# B&R Automation Studio project NAEUL004C00R13L518F00 (part 33)

#### Act_Main.st - Do Not Change!!!
```iecst
(** 2020-10-05 **)
ACTION Act_Main:
	//Reset Done
	IF tylocalHWInfo.Out.eStatus = Done AND tylocalHWInfo.In.eAct = HWInfoActIdle THEN
		tylocalHWInfo.Out.eStat	:= HWInfoActIdle;
	END_IF

	//Set tylocalHWInfo.In.eAct
	IF tylocalHWInfo.Out.eStatus = Idle THEN
		tylocalHWInfo.Out.eStat	:= tylocalHWInfo.In.eAct;
	END_IF

	//Main
	CASE tylocalHWInfo.Out.eStat OF

		HWInfoActIdle:
			IF tylocalHWInfo.Out.eStatus <> Idle THEN	//Reset Data
				//Private
				fbGetIPAddr(enable := FALSE);
				fbGetMacAddr(enable := FALSE);
				fbSetIPAddr(enable := FALSE);
				fbSetSubnetMask(enable := FALSE);
				fbGetETHConfigMode(enable := FALSE);
				fbSetETHConfigMode(enable := FALSE);

				tylocalHWInfo.Out.sStatTxt	:= a_sStatText[tylocalHWInfo.Out.eStat];

			END_IF

			tylocalHWInfo.Out.eStatus	:= Idle;

		HWInfoActGetIPAddr:
			IF tylocalHWInfo.Out.eStatus = Idle OR tylocalHWInfo.Out.eStatus = Busy THEN

				tylocalHWInfo.Out.eStatus	:= Busy;

				tylocalHWInfo.Out.sStatTxt	:= a_sStatText[tylocalHWInfo.Out.eStat];

				IF DiagCpuIsSimulated() = FALSE THEN
					fbGetIPAddr(enable := TRUE);
					IF fbGetIPAddr.status = 0 THEN
						tylocalHWInfo.Out.eStatus	:= Done;
					ELSIF fbGetIPAddr.status < 65534 THEN
						udiStatus	:= 10000;	//Get IP Address Error
						tylocalHWInfo.Out.eStatus		:= Error;
					END_IF

				ELSE
					tylocalHWInfo.Out.eStatus	:= Done;
					tylocalHWInfo.Out.sIPAddr	:= '127.0.0.1';

				END_IF

			END_IF

		HWInfoActGetSubnetMask:
			IF tylocalHWInfo.Out.eStatus = Idle OR tylocalHWInfo.Out.eStatus = Busy THEN

				tylocalHWInfo.Out.eStatus	:= Busy;

				tylocalHWInfo.Out.sStatTxt	:= a_sStatText[tylocalHWInfo.Out.eStat];

				IF DiagCpuIsSimulated() = FALSE THEN
					fbGetSubnetMask(enable := TRUE);
					IF fbGetSubnetMask.status = 0 THEN
						tylocalHWInfo.Out.eStatus	:= Done;
					ELSIF fbGetSubnetMask.status < 65534 THEN
						udiStatus	:= 10001;	//Get Subnet Mask Error
						tylocalHWInfo.Out.eStatus		:= Error;
					END_IF

				ELSE
					tylocalHWInfo.Out.eStatus		:= Done;
					tylocalHWInfo.Out.sSubnetMask	:= '255.255.0.0';

				END_IF

			END_IF

		HWInfoActGetMacAddr:
			IF tylocalHWInfo.Out.eStatus = Idle OR tylocalHWInfo.Out.eStatus = Busy THEN

				tylocalHWInfo.Out.eStatus	:= Busy;

				tylocalHWInfo.Out.sStatTxt	:= a_sStatText[tylocalHWInfo.Out.eStat];

				IF DiagCpuIsSimulated() = FALSE THEN
					fbGetMacAddr(enable := TRUE);
					IF fbGetMacAddr.status = 0 THEN
						tylocalHWInfo.Out.eStatus	:= Done;
					ELSIF fbGetMacAddr.status < 65534 THEN
						udiStatus	:= 10002;	//Get Mac Address Error
						tylocalHWInfo.Out.eStatus		:= Error;
					END_IF

				ELSE
					tylocalHWInfo.Out.eStatus	:= Done;

				END_IF

			END_IF

		HWInfoActSetIPAddr:
			IF tylocalHWInfo.Out.eStatus = Idle OR tylocalHWInfo.Out.eStatus = Busy THEN

				tylocalHWInfo.Out.eStatus	:= Busy;

				tylocalHWInfo.Out.sStatTxt	:= a_sStatText[tylocalHWInfo.Out.eStat];

				IF DiagCpuIsSimulated() = FALSE THEN
					fbSetIPAddr(enable := TRUE);
					IF fbSetIPAddr.status = 0 THEN
						tylocalHWInfo.Out.sIPAddr	:= p_sSetIPAddr;
						tylocalHWInfo.Out.eStatus	:= Done;
					ELSIF fbSetIPAddr.status < 65534 THEN
						udiStatus	:= 10003;	//Set IP Address Error
						tylocalHWInfo.Out.eStatus		:= Error;
					END_IF

				ELSE
					tylocalHWInfo.Out.eStatus	:= Done;

				END_IF

			END_IF

		HWInfoActSetSubnetMask:
			IF tylocalHWInfo.Out.eStatus = Idle OR tylocalHWInfo.Out.eStatus = Busy THEN

				tylocalHWInfo.Out.eStatus	:= Busy;

				tylocalHWInfo.Out.sStatTxt	:= a_sStatText[tylocalHWInfo.Out.eStat];

				IF DiagCpuIsSimulated() = FALSE THEN
					fbSetSubnetMask(enable := TRUE);
					IF fbSetSubnetMask.status = 0 THEN
						tylocalHWInfo.Out.sSubnetMask	:= p_sSetSubnetMask;
						tylocalHWInfo.Out.eStatus		:= Done;
					ELSIF fbSetSubnetMask.status < 65534 THEN
						udiStatus	:= 10004;	//Set Subnet Mask Error
						tylocalHWInfo.Out.eStatus		:= Error;
					END_IF

				ELSE
					tylocalHWInfo.Out.eStatus	:= Done;

				END_IF

			END_IF

		HWInfoActGetEthConfigMode:
			IF tylocalHWInfo.Out.eStatus = Idle OR tylocalHWInfo.Out.eStatus = Busy THEN

				tylocalHWInfo.Out.eStatus	:= Busy;

				tylocalHWInfo.Out.sStatTxt	:= a_sStatText[tylocalHWInfo.Out.eStat];
				IF DiagCpuIsSimulated() = FALSE THEN
					fbGetETHConfigMode(enable := TRUE);
					IF fbGetETHConfigMode.status = 0 THEN
						tylocalHWInfo.Out.udiConfigMode := fbGetETHConfigMode.ConfigMode;
						tylocalHWInfo.Out.eStatus	:= Done;
					ELSIF fbGetETHConfigMode.status < 65534 THEN
						udiStatus	:= 10005;	//Get Network Configuration  Error
						tylocalHWInfo.Out.eStatus		:= Error;
					END_IF

				ELSE
					tylocalHWInfo.Out.eStatus	:= Done;

				END_IF

			END_IF

		HWInfoActSetEthConfigMode:
			IF tylocalHWInfo.Out.eStatus = Idle OR tylocalHWInfo.Out.eStatus = Busy THEN

				tylocalHWInfo.Out.eStatus	:= Busy;

				tylocalHWInfo.Out.sStatTxt	:= a_sStatText[tylocalHWInfo.Out.eStat];

				IF DiagCpuIsSimulated() = FALSE THEN
					fbSetETHConfigMode.ConfigMode := USINT_TO_UDINT(p_usiNetworkMod);
					fbSetETHConfigMode(enable := TRUE);

					IF fbSetETHConfigMode.status = 0 THEN
						tylocalHWInfo.Out.eStatus	:= Done;
					ELSIF fbSetETHConfigMode.status < 65534 THEN
						udiStatus	:= 10006;	//Set Network Configuration  Error
						tylocalHWInfo.Out.eStatus		:= Error;
					END_IF

				ELSE
					tylocalHWInfo.Out.eStatus	:= Done;

				END_IF

			END_IF

		HWInfoActSetDefaultGateway:
			IF tylocalHWInfo.Out.eStatus = Idle OR tylocalHWInfo.Out.eStatus = Busy THEN

				tylocalHWInfo.Out.eStatus	:= Busy;

				tylocalHWInfo.Out.sStatTxt	:= a_sStatText[tylocalHWInfo.Out.eStat];

				IF DiagCpuIsSimulated() = FALSE THEN
					fbSetDefaultGateway.pGateway := ADR(p_sSetDefaultGW);
					fbSetDefaultGateway(enable := TRUE);

					IF fbSetDefaultGateway.status = 0 THEN
						tylocalHWInfo.Out.eStatus	:= Done;
					ELSIF fbSetDefaultGateway.status < 65534 THEN
						udiStatus	:= 10007;	//'Set Default Gateway IP Error'
						tylocalHWInfo.Out.eStatus		:= Error;
					END_IF

				ELSE
					tylocalHWInfo.Out.eStatus	:= Done;
				END_IF

			END_IF

	END_CASE

	//Generate file
//	IF tylocalHWInfo.Out.a_usiMacAddr[3] <> 0 AND usiInitialFile <2 THEN
//		CASE usi OF
//			0:
//				FOR usi:= 0 TO 5 DO
//					//a_sMacAddr[usi] := USINT_TO_STRING(tylocalHWInfo.Out.a_usiMacAddr[usi]);
//					sprintf1(ADR(a_sMacAddr[usi]), ADR('%+02x'), tylocalHWInfo.Out.a_usiMacAddr[usi]);
//				END_FOR
//				sMacAddr := CONCAT('PLC= ',CONCAT(a_sMacAddr[0],'-'));
//				FOR usi := 1 TO 5 DO
//					sMacAddr := CONCAT(CONCAT(sMacAddr,a_sMacAddr[usi]),'-');
//				END_FOR
//				sMacAddr := DELETE(sMacAddr,1,LEN(sMacAddr));
//				usi := 1;
//			1:
//				fbFileFullWrite_0(bEn := TRUE, sDevice := 'Log', sFile := 'PLC_MacAddress.txt', udiOffset := 0, p_Src := ADR(sMacAddr), udiLen := SIZEOF(sMacAddr), udiOption := 0);
//				IF fbFileFullWrite_0.udiStatus = 0 THEN
//					fbFileFullWrite_0(bEn := FALSE);
//					IF usiInitialFile = 1 THEN
//						usi := 0;
//					END_IF
//					usiInitialFile := usiInitialFile +1;
//				END_IF
//
//		END_CASE
//	END_IF
END_ACTION
```

#### Act_Alarm.st - Do Not Change!!!
```iecst
(** 2019-03-25 **)
ACTION Act_Alarm:
	IF tylocalHWInfo.In.udiRstErr <> udiRstErrOld THEN
		bRstErr			:= TRUE;
		udiRstErrOld	:= tylocalHWInfo.In.udiRstErr;
	ELSE
		bRstErr			:= FALSE;
	END_IF

	//Reset Error
	IF (tylocalHWInfo.Out.eStatus = Error) AND bRstErr THEN
		tylocalHWInfo.In.eAct	:= HWInfoActIdle;
		tylocalHWInfo.Out.eStat	:= HWInfoActIdle;
	END_IF

	//Error
	IF EDGEPOS(tylocalHWInfo.Out.eStatus = Error) THEN

		tylocalHWInfo.Out.tyAlmData.udiCode			:= udiStatus;
		tylocalHWInfo.Out.tyAlmData.eSeverity		:= AlmSeverityError;
		tylocalHWInfo.Out.tyAlmData.udiRunTime		:= tylocalHWInfo.Out.tyAlmData.udiRunTime + 1;
		tylocalHWInfo.Out.tyAlmData.bAlm			:= TRUE;
		tylocalHWInfo.Out.tyAlmData.udiModuleNum	:= udiModuleNum;
		g_tyAlmProgNm.sHWinfoProgNm					:= tylocalHWInfo.In.sProgNm;

	ELSIF bRstErr AND (tylocalHWInfo.Out.tyAlmData.udiCode <> 0) THEN

		tylocalHWInfo.Out.tyAlmData.udiCode		:= 0;
		tylocalHWInfo.Out.tyAlmData.eSeverity	:= AlmSeverityNA;
		tylocalHWInfo.Out.tyAlmData.bAlm		:= FALSE;

		tylocalHWInfo.Out.sStatTxt	:= a_sStatText[tylocalHWInfo.Out.eStat];

	END_IF

END_ACTION
```

#### Local.var - Do Not Change!!!
```iecst
(*2020-09-22*)
VAR
	tylocalHWInfo : tyHWInfo;
END_VAR
(**)
(*Local Action, State & Status*)
VAR
	eStatus : eFBStatus := Idle;
	udiStatus : UDINT := 0;
	sStatTxt : STRING[200] := '';
	a_sStatText : ARRAY[0..50] OF STRING[200] := ['Idling','Get IP Address','Get IP Subnet Mask','Get Mac Address','Setting IP Address','Setting IP Subnet Mask',45('')];
END_VAR
(**)
(*Local Alarm*)
VAR
	tyAlmData : tyAlmDat;
	a_tyAlmText : ARRAY[10000..10099] OF tyAlmTxt := [(sAlmText:='Get IP Address Error',sRcyText:='Failed To Obtain The IP Address. Please Contact Nutek For A Possible Solution.'),(sAlmText:='Get Subnet Mask Error',sRcyText:='Failed To Obtain The Subnet Mask. Please Contact Nutek For A Possible Solution.'),(sAlmText:='Get Mac Address Error',sRcyText:='Failed To Obtain The Mac Address. Please Contact Nutek For A Possible Solution.'),(sAlmText:='Set IP Address Error',sRcyText:='Invalid IP Address Configuration. Please Contact Nutek For A Possible Solution.'),(sAlmText:='Set Subnet Mask Error',sRcyText:='Invalid Subnet Mask Configuration. Please Contact Nutek For A Possible Solution.'),(sAlmText:='Get Network Configuration Mode Error',sRcyText:='Failed To Obtain The Network Configuration. Please Contact Nutek For A Possible Solution.'),(sAlmText:='Set Network Configuration Mode Error',sRcyText:='Invalid Network Configuration . Please Contact Nutek For A Possible Solution.'),(sAlmText:='Set Default Gateway IP Error',sRcyText:='Invalid IP Address Configuration. Please Contact Nutek For A Possible Solution.'),92((0))];
END_VAR
(**)
(*Local Output*)
VAR
	sIPAddr : STRING[15];
	sSubnetMask : STRING[15];
	a_usiMacAddr : ARRAY[0..5] OF USINT;
	udiConfigMode : UDINT;
END_VAR
(**)
(*Local Input*)
VAR
	udiRstErr : UDINT := 0;
	sSetIPAddr : STRING[15];
	sSetSubnetMask : STRING[15];
	sDevice : STRING[3] := 'IF2';
	sProgNm : STRING[15] := 'HWInfo';
	bNtSettingsLoadDone : BOOL := TRUE;
	usiNetworkMode : USINT;
	sSetDefaultGW : STRING[15];
END_VAR
(**)
(*Local*)
VAR
	bRstErr : BOOL;
	udiRstErrOld : UDINT;
	bInitDone : BOOL;
	bInitialDone : BOOL;
	fbGetIPAddr : CfgGetIPAddr;
	fbGetSubnetMask : CfgGetSubnetMask;
	fbGetMacAddr : CfgGetMacAddr;
	fbSetIPAddr : CfgSetIPAddr;
	fbSetSubnetMask : CfgSetSubnetMask;
	fbSetETHConfigMode : CfgSetEthConfigMode;
	fbGetETHConfigMode : CfgGetEthConfigMode;
	fbSetDefaultGateway : CfgSetDefaultGateway;
	udiModuleNum : UDINT := 5651;
END_VAR
(**)
(*MAC Address*)
VAR
	sMacAddress : tysMacAddress;
END_VAR
(**)
VAR
	sPLCMacAddress : STRING[27];
	sHMIMacAddress : STRING[27];
END_VAR
```

#### InputRef.var - not listed in the package file held
```iecst
(*2020-09-22*)
(**)
(*General*)
VAR
	p_eAct : REFERENCE TO eHWInfoAction;
	p_udiRstErr : REFERENCE TO UDINT;
END_VAR
(**)
(*Configuration*)
VAR
	p_sSetIPAddr : REFERENCE TO STRING[15];
	p_sSetSubnetMask : REFERENCE TO STRING[15];
	p_sDevice : REFERENCE TO STRING[3];
	p_sProgNm : REFERENCE TO STRING[15];
	p_bNtSettingsLoadDone : REFERENCE TO BOOL;
	p_usiNetworkMod : REFERENCE TO USINT;
	p_sSetDefaultGW : REFERENCE TO STRING[15];
END_VAR
```

#### InputRef_Link.var - not listed in the package file held
```iecst
(*2019-03-25*)
(**)
VAR
	p_bLinkStartupRun : REFERENCE TO BOOL;
	p_sHMIMacAdd : REFERENCE TO STRING[27];
END_VAR
```

#### Act_InitGlobal.st - not listed in the package file held
```iecst
(** 2020-09-22 **)
ACTION Act_InitGlobal:

	(* Always Change If Project Change *)

	//Pass Data To Link
	p_bLinkStartupRun ACCESS p_StartupRun;

	//Pass Data To Internal Use
	p_udiRstErr ACCESS p_RstErrReset;
	p_sSetIPAddr ACCESS p_UISetIPAddr;
	p_sSetSubnetMask ACCESS p_UISetSubnetMask;
	p_sDevice ACCESS p_NtParamHWInfoDevice;
	p_sProgNm ACCESS p_NtParamHWInfoProgNm;
	p_bNtSettingsLoadDone ACCESS p_StartupNtSettingsLoadDone;
	p_usiNetworkMod ACCESS p_UINetworkMode;

	//HMI MAC Address
	p_sHMIMacAdd ACCESS p_NtParamHWInfoHMIMacAddress;
	p_sSetDefaultGW ACCESS p_McParamDefaultGateway;

	(* Always Change If Project Change *)

END_ACTION
```

#### Act_InitLocal.st - not listed in the package file held
```iecst
(** 2020-09-22 **)
ACTION Act_InitLocal:

	//Input Reference Link To Local Variable
	p_eAct ACCESS ADR(eAct);
	p_udiRstErr ACCESS ADR(udiRstErr);
	p_sSetIPAddr ACCESS ADR(sSetIPAddr);
	p_sSetSubnetMask ACCESS ADR(sSetSubnetMask);
	p_sDevice ACCESS ADR(sDevice);
	p_sProgNm ACCESS ADR(sProgNm);
	p_bNtSettingsLoadDone ACCESS ADR(bNtSettingsLoadDone);
	p_usiNetworkMod ACCESS ADR(usiNetworkMode);
	p_sSetDefaultGW ACCESS ADR(sSetDefaultGW);
END_ACTION
```

### TLBuz.typ - Do Not Change!!!
```iecst
(*2020-02-19*)
(**)
(*Action*)

TYPE
	eTLBuzAction :
		(
		TLBuzActIdle,
		TLBuzActSetGreen,
		TLBuzActSetWhite,
		TLBuzActSetRed,
		TLBuzActSetAmber,
		TLBuzActSetBlue,
		TLBuzActSetBuz,
		TLBuzActRstGreen,
		TLBuzActRstWhite,
		TLBuzActRstRed,
		TLBuzActRstAmber,
		TLBuzActRstBlue,
		TLBuzActRstBuz,
		TLBuzActSetAll,
		TLBuzActRstAll
		);
	eTLBuzMod :
		(
		TLBuzModNutek,
		TLBuzModAptiv,
		TLBuzModMEK,
		TLBuzModBHTC,
		TLBuzModSiemens_2Colour
		);
	tyTLBuz : 	STRUCT
		In : tyTLBuzIn1;
		Out : tyTLBuzOut1;
	END_STRUCT;
	tyTLBuzIn1 : 	STRUCT
		eAct : eTLBuzAction; (*Tower Light Buzzer's Action*)
		bCoverSwitchSig : BOOL := FALSE; (*Cover Switch Signal*)
		bAOIErrSig : BOOL := FALSE; (*AOI Err Signal*)
		bAOIOriginSig : BOOL := FALSE; (*AOI Origin Signal*)
		bBuzAlertEn : BOOL := FALSE; (*Buzzer Alert Enable*)
		bTLBlueFlashEn : BOOL := FALSE; (*Tower Light Blue Flash Enable*)
		bTLAmberFlashEn : BOOL := FALSE; (*Tower Light Amber Flash Enable*)
		bTLWhiteFlashEn : BOOL := FALSE; (*Tower Light White Flash Enable*)
		bTLRedFlashEn : BOOL := FALSE; (*Tower Light Red Flash Enable*)
		bTLGreenFlashEn : BOOL := FALSE; (*Tower Light Green Flash Enable*)
		bUIManualMod : BOOL := FALSE; (*Manual Mode*)
		bStartup : BOOL := FALSE; (*Startup Mode*)
		bErr : BOOL := FALSE; (*Error Exist*)
		bErrNoBuz : BOOL := FALSE; (*Error Exist With No Buzzer*)
		bWarning : ARRAY[0..5]OF BOOL := [6(FALSE)]; (*Warning*)
		bWarningNoBuz : ARRAY[0..5]OF BOOL := [6(FALSE)]; (*Warning With No Buzzer*)
		bChgRcp : BOOL := FALSE; (*Change Recipe*)
		bSeqStop : BOOL := FALSE; (*Sequence Stop*)
		bStep : BOOL := FALSE; (*Step*)
		bOps : BOOL := FALSE; (*Operation Mode*)
		bStandby : BOOL := FALSE; (*Standby Mode*)
		bSimulation : BOOL := FALSE; (*Simulation Mode*)
		bMuteBuz : BOOL := FALSE; (*Mute Buzzer*)
		tTLChgRcpBlinkTm : TIME := T#200ms; (*Tower Light Change Recipe Blink Timer*)
		tTLErrBlinkTm : TIME := T#500ms; (*Tower Light Error Blink Timer*)
		tBuzErrOnTm : TIME := T#500ms; (*Buzzer Error On Timer*)
		tBuzErrRestTm : TIME := T#500ms; (*Buzzer Error Reset Timer*)
		usiBuzErrOnCntr : USINT := 3; (*Buzzer Error On Counter*)
		bBuzErrStopSeqEn : BOOL := FALSE; (*Buzzer Error Stop Sequence Timer Counter*)
		usiBuzErrStopSeqCntr : USINT := 3; (*Buzzer Error Stop Sequence Counter*)
		tTLWarnBlinkTm : ARRAY[0..5]OF TIME := [6(T#500ms)]; (*Tower Light Warning Blink Timer*)
		tBuzWarnOnTm : ARRAY[0..5]OF TIME := [6(T#500ms)]; (*Buzzer Warning On Timer*)
		tBuzWarnRestTm : ARRAY[0..5]OF TIME := [6(T#5s)]; (*Buzzer Warning Reset Timer*)
		usiBuzWarnOnCntr : ARRAY[0..5]OF USINT := [6(3)]; (*Buzzer Warning On Counter*)
		bBuzWarnStopSeqEn : ARRAY[0..5]OF BOOL := [6(FALSE)]; (*Buzzer Warning Stop Sequence Enable*)
		usiBuzWarnStopSeqCntr : ARRAY[0..5]OF USINT := [6(3)]; (*Buzzer Warning Stop Sequence Counter*)
		tTLWarn1BlinkTm : TIME := T#500ms;
		tBuzWarn1OnTm : TIME := T#500ms;
		tBuzWarn1RestTm : TIME := T#5s;
		usiBuzWarn1OnCntr : USINT := 3;
		bBuzWarn1StopSeqEn : BOOL := FALSE;
		usiBuzWarn1StopSeqCntr : USINT := 3;
		tTLWarn2BlinkTm : TIME := T#500ms;
		tBuzWarn2OnTm : TIME := T#500ms;
		tBuzWarn2RestTm : TIME := T#5s;
		usiBuzWarn2OnCntr : USINT := 3;
		bBuzWarn2StopSeqEn : BOOL := FALSE;
		usiBuzWarn2StopSeqCntr : USINT := 3;
		tTLWarn3BlinkTm : TIME := T#500ms;
		tBuzWarn3OnTm : TIME := T#500ms;
		tBuzWarn3RestTm : TIME := T#5s;
		usiBuzWarn3OnCntr : USINT := 3;
		bBuzWarn3StopSeqEn : BOOL := FALSE;
		usiBuzWarn3StopSeqCntr : USINT := 3;
		tTLWarn4BlinkTm : TIME := T#500ms;
		tBuzWarn4OnTm : TIME := T#500ms;
		tBuzWarn4RestTm : TIME := T#5s;
		usiBuzWarn4OnCntr : USINT := 3;
		bBuzWarn4StopSeqEn : BOOL := FALSE;
		usiBuzWarn4StopSeqCntr : USINT := 3;
		tTLWarn5BlinkTm : TIME := T#500ms;
		tBuzWarn5OnTm : TIME := T#500ms;
		tBuzWarn5RestTm : TIME := T#5s;
		usiBuzWarn5OnCntr : USINT := 3;
		bBuzWarn5StopSeqEn : BOOL := FALSE;
		usiBuzWarn5StopSeqCntr : USINT := 3;
		tBuzAlertOnTm : TIME := T#500ms; (*Buzzer Alert On Timer*)
		tBuzAlertRestTm : TIME := T#5s; (*Buzzer Alert Reset Timer*)
		usiBuzAlertOnCntr : USINT := 3; (*Buzzer Alert On Counter*)
		bBuzAlertStopSeqEn : BOOL := FALSE; (*Buzzer Alert Stop Sequence Enable*)
		usiBuzAlertStopSeqCntr : USINT := 3; (*Buzzer Alert Stop Sequence Counter*)
		tTLBlueBlinkTm : TIME := T#500ms; (*Tower Light Blue Blink Timer*)
		tTLAmberBlinkTm : TIME := T#500ms; (*Tower Light Amber Blink Timer*)
		tTLWhiteBlinkTm : TIME := T#500ms; (*Tower Light White Blink Timer*)
		tTLRedBlinkTm : TIME := T#500ms; (*Tower Light Red Blink Timer*)
		tTLGreenBlinkTm : TIME := T#500ms; (*Tower Light Green Blink Timer*)
		eTLBuzMode : eTLBuzMod := TLBuzModNutek; (*Tower Light Buzzer Mode*)
		bMcParamAGVComEn : BOOL;
		eMcParamMagExMode : eMcMagExchangeMode;
	END_STRUCT;
	tyTLBuzOut1 : 	STRUCT
		eStat : eTLBuzAction := TLBuzActIdle; (*Tower Light Buzzer's State*)
		eStatus : eFBStatus := Idle; (*Tower Light Buzzer's Status*)
		sStatTxt : STRING[200] := ''; (*Tower Light Buzzer's State in Text*)
		bTLBlue : BOOL; (*Tower Light Blue*)
		bTLRed : BOOL; (*Tower Light Red*)
		bTLAmber : BOOL; (*Tower Light Amber*)
		bTLWhite : BOOL; (*Tower Light White*)
		bTLGreen : BOOL; (*Tower Light Green*)
		bBuzBeep : BOOL; (*Buzzer Beeping*)
	END_STRUCT;
END_TYPE
```

### TLBuz.var - Change By Project
```iecst
(*2019-03-25*)
VAR
	g_tyTLBuz : tyTLBuzOut1;
END_VAR
(**)
```

### Program Logical/TLBuz/TLBuz (IEC, version 1.00.0) - 1.00.0 - NtTLBuz v5.00.0

#### Act_InputConfig.st - Change By Project
```iecst
ACTION Act_InputConfig:

	tylocalTLBuz.In.bStartup 					:= g_tyStartUp.bRun;
	tylocalTLBuz.In.bErr	 					:= g_tyAlm.bErr;
	tylocalTLBuz.In.bSeqStop    				:= g_tyOps.bStatusCycleStop;
	tylocalTLBuz.In.bStep						:= g_tyOps.bStatusStep;
	tylocalTLBuz.In.bOps						:= g_tyOps.bStatusRun;
	tylocalTLBuz.In.bStandby					:= g_tyOps.bStatusStop;
	tylocalTLBuz.In.bMuteBuz					:= g_tyUIOut.bUIMuteBuz;
	tylocalTLBuz.In.bUIManualMod				:= g_tyUIOut.bUIManualMod;

	//  -----------------------------------------  TLBuz 5.00.2  -----------------------------------------	//

	tylocalTLBuz.In.tTLChgRcpBlinkTm 			:= g_tyNtParamCurr.tyTLBuz.tTLChgRcpBlinkTm;
	tylocalTLBuz.In.tTLErrBlinkTm	 			:= g_tyNtParamCurr.tyTLBuz.tTLErrBlinkTm;
	tylocalTLBuz.In.tBuzErrOnTm		 			:= g_tyNtParamCurr.tyTLBuz.tBuzErrOnTm;
	tylocalTLBuz.In.tBuzErrRestTm	 			:= g_tyNtParamCurr.tyTLBuz.tBuzErrRestTm;
	tylocalTLBuz.In.usiBuzAlertOnCntr			:= g_tyNtParamCurr.tyTLBuz.usiBuzErrOnCntr;
	tylocalTLBuz.In.bBuzErrStopSeqEn			:= g_tyNtParamCurr.tyTLBuz.bBuzErrStopSeqEn;
	tylocalTLBuz.In.usiBuzErrStopSeqCntr 		:= g_tyNtParamCurr.tyTLBuz.usiBuzErrStopSeqCntr;

	tylocalTLBuz.In.tTLWarnBlinkTm  			:= g_tyNtParamCurr.tyTLBuz.tTLWarnBlinkTm;
	tylocalTLBuz.In.tBuzWarnOnTm				:= g_tyNtParamCurr.tyTLBuz.tBuzWarnOnTm;
	tylocalTLBuz.In.tBuzWarnRestTm				:= g_tyNtParamCurr.tyTLBuz.tBuzWarnRestTm;
	tylocalTLBuz.In.usiBuzWarnOnCntr			:= g_tyNtParamCurr.tyTLBuz.usiBuzWarnOnCntr;
	tylocalTLBuz.In.bBuzWarnStopSeqEn			:= g_tyNtParamCurr.tyTLBuz.bBuzWarnStopSeqEn;
	tylocalTLBuz.In.usiBuzWarnStopSeqCntr		:= g_tyNtParamCurr.tyTLBuz.usiBuzWarnStopSeqCntr;

	tylocalTLBuz.In.tTLWarn1BlinkTm  			:= g_tyNtParamCurr.tyTLBuz.tTLWarn1BlinkTm;
	tylocalTLBuz.In.tBuzWarn1OnTm				:= g_tyNtParamCurr.tyTLBuz.tBuzWarn1OnTm;
	tylocalTLBuz.In.tBuzWarn1RestTm				:= g_tyNtParamCurr.tyTLBuz.tBuzWarn1RestTm;
	tylocalTLBuz.In.usiBuzWarn1OnCntr			:= g_tyNtParamCurr.tyTLBuz.usiBuzWarn1OnCntr;
	tylocalTLBuz.In.bBuzWarn1StopSeqEn			:= g_tyNtParamCurr.tyTLBuz.bBuzWarn1StopSeqEn;
	tylocalTLBuz.In.usiBuzWarn1StopSeqCntr		:= g_tyNtParamCurr.tyTLBuz.usiBuzWarn1StopSeqCntr;

	tylocalTLBuz.In.tTLWarn2BlinkTm  			:= g_tyNtParamCurr.tyTLBuz.tTLWarn2BlinkTm;
	tylocalTLBuz.In.tBuzWarn2OnTm				:= g_tyNtParamCurr.tyTLBuz.tBuzWarn2OnTm;
	tylocalTLBuz.In.tBuzWarn2RestTm				:= g_tyNtParamCurr.tyTLBuz.tBuzWarn2RestTm;
	tylocalTLBuz.In.usiBuzWarn2OnCntr			:= g_tyNtParamCurr.tyTLBuz.usiBuzWarn2OnCntr;
	tylocalTLBuz.In.bBuzWarn2StopSeqEn			:= g_tyNtParamCurr.tyTLBuz.bBuzWarn2StopSeqEn;
	tylocalTLBuz.In.usiBuzWarn2StopSeqCntr		:= g_tyNtParamCurr.tyTLBuz.usiBuzWarn2StopSeqCntr;

	tylocalTLBuz.In.tTLWarn3BlinkTm  			:= g_tyNtParamCurr.tyTLBuz.tTLWarn3BlinkTm;
	tylocalTLBuz.In.tBuzWarn3OnTm				:= g_tyNtParamCurr.tyTLBuz.tBuzWarn3OnTm;
	tylocalTLBuz.In.tBuzWarn3RestTm				:= g_tyNtParamCurr.tyTLBuz.tBuzWarn3RestTm;
	tylocalTLBuz.In.usiBuzWarn3OnCntr			:= g_tyNtParamCurr.tyTLBuz.usiBuzWarn3OnCntr;
	tylocalTLBuz.In.bBuzWarn3StopSeqEn			:= g_tyNtParamCurr.tyTLBuz.bBuzWarn3StopSeqEn;
	tylocalTLBuz.In.usiBuzWarn3StopSeqCntr		:= g_tyNtParamCurr.tyTLBuz.usiBuzWarn3StopSeqCntr;

	tylocalTLBuz.In.tTLWarn4BlinkTm  			:= g_tyNtParamCurr.tyTLBuz.tTLWarn4BlinkTm;
	tylocalTLBuz.In.tBuzWarn4OnTm				:= g_tyNtParamCurr.tyTLBuz.tBuzWarn4OnTm;
	tylocalTLBuz.In.tBuzWarn4RestTm				:= g_tyNtParamCurr.tyTLBuz.tBuzWarn4RestTm;
	tylocalTLBuz.In.usiBuzWarn4OnCntr			:= g_tyNtParamCurr.tyTLBuz.usiBuzWarn4OnCntr;
	tylocalTLBuz.In.bBuzWarn4StopSeqEn			:= g_tyNtParamCurr.tyTLBuz.bBuzWarn4StopSeqEn;
	tylocalTLBuz.In.usiBuzWarn4StopSeqCntr		:= g_tyNtParamCurr.tyTLBuz.usiBuzWarn4StopSeqCntr;

	tylocalTLBuz.In.tTLWarn5BlinkTm  			:= g_tyNtParamCurr.tyTLBuz.tTLWarn5BlinkTm;
	tylocalTLBuz.In.tBuzWarn5OnTm				:= g_tyNtParamCurr.tyTLBuz.tBuzWarn5OnTm;
	tylocalTLBuz.In.tBuzWarn5RestTm				:= g_tyNtParamCurr.tyTLBuz.tBuzWarn5RestTm;
	tylocalTLBuz.In.usiBuzWarn5OnCntr			:= g_tyNtParamCurr.tyTLBuz.usiBuzWarn5OnCntr;
	tylocalTLBuz.In.bBuzWarn5StopSeqEn			:= g_tyNtParamCurr.tyTLBuz.bBuzWarn5StopSeqEn;
	tylocalTLBuz.In.usiBuzWarn5StopSeqCntr		:= g_tyNtParamCurr.tyTLBuz.usiBuzWarn5StopSeqCntr;

	tylocalTLBuz.In.tBuzAlertOnTm 				:= g_tyNtParamCurr.tyTLBuz.tBuzAlertOnTm;
	tylocalTLBuz.In.tBuzAlertRestTm 			:= g_tyNtParamCurr.tyTLBuz.tBuzAlertRestTm;
	tylocalTLBuz.In.usiBuzAlertOnCntr 			:= g_tyNtParamCurr.tyTLBuz.usiBuzAlertOnCntr;
	tylocalTLBuz.In.bBuzAlertStopSeqEn  		:= g_tyNtParamCurr.tyTLBuz.bBuzAlertStopSeqEn;
	tylocalTLBuz.In.usiBuzAlertStopSeqCntr		:= g_tyNtParamCurr.tyTLBuz.usiBuzAlertStopSeqCntr;

	tylocalTLBuz.In.tTLBlueBlinkTm				:= g_tyNtParamCurr.tyTLBuz.tTLBlueBlinkTm;
	tylocalTLBuz.In.tTLAmberBlinkTm				:= g_tyNtParamCurr.tyTLBuz.tTLAmberBlinkTm;
	tylocalTLBuz.In.tTLWhiteBlinkTm				:= g_tyNtParamCurr.tyTLBuz.tTLWhiteBlinkTm;
	tylocalTLBuz.In.tTLRedBlinkTm				:= g_tyNtParamCurr.tyTLBuz.tTLRedBlinkTm;
	tylocalTLBuz.In.tTLGreenBlinkTm				:= g_tyNtParamCurr.tyTLBuz.tTLGreenBlinkTm;

	//  ----------------------------------------------  ||  ---------------------------------------------	//
	tylocalTLBuz.In.eTLBuzMode					:= g_tyNtParamCurr.tyTLBuz.eTLBuzMode;
	tylocalTLBuz.In.bCoverSwitchSig				:= g_tyDInput.bCoverSWSig;

	tylocalTLBuz.In.bMcParamAGVComEn			:= g_tyMcParamCurr.bAGVComEn;
	tylocalTLBuz.In.eMcParamMagExMode			:= g_tyMcParamCurr.eMagExMode;

	tylocalTLBuz.In.bWarning[0]					:= g_tyAlm.bWarning OR (g_tyAlm.bInfo AND NOT (g_tyAlm.bInfoLF AND g_tyMcParamCurr.bLFBuzMute)AND NOT(g_tyOpsMagConv1.bMagFullInfo AND g_tyOpsMagConv1.bTLMuteBuzzer) );
	tylocalTLBuz.In.bWarningNoBuz[0]			:= (g_tyAlm.bInfoLF AND g_tyMcParamCurr.bLFBuzMute) OR (g_tyOpsMagConv1.bMagFullInfo AND g_tyOpsMagConv1.bTLMuteBuzzer );

	IF g_tyUIOut.bUIManualMod THEN
		tylocalTLBuz.In.eAct	:= g_tyUIOut.eMnlAct.eTLBuzAct;
	ELSE
		tylocalTLBuz.In.eAct	:= tylocalTLBuz.In.eAct;
	END_IF

END_ACTION
```

#### Act_OutputConfig.st - Change By Project
```iecst
ACTION Act_OutputConfig:

 g_tyTLBuz := tylocalTLBuz.Out;

END_ACTION
```

#### Cyclic.st - Do Not Change!!!
```iecst
(** 2020-03-16 **)
PROGRAM _CYCLIC

	IF bInitialDone = FALSE THEN
		bInitialDone	:= TRUE;

		Act_Initial;

	ELSE

		Act_InputConfig;
		Act_Main;

		CASE p_eTLBuzMode OF
			TLBuzModNutek:
				Act_Background;
			TLBuzModAptiv:
				Act_Background1;
			TLBuzModMEK:
				Act_Background2;
			TLBuzModBHTC:
				Act_Background3;
			TLBuzModSiemens_2Colour:
				Act_Background4;

		END_CASE
		Act_OutputConfig;
	END_IF

END_PROGRAM
```

#### Act_Main.st - Do Not Change!!!
```iecst
(** 2020-02-18 **)
ACTION Act_Main:
		//Set p_eAct
	IF tylocalTLBuz.Out.eStatus = Idle OR tylocalTLBuz.Out.eStatus = Busy OR tylocalTLBuz.Out.eStatus = Done THEN
		tylocalTLBuz.Out.eStat	:= tylocalTLBuz.In.eAct;
	END_IF
	IF eStatOld <> tylocalTLBuz.Out.eStat THEN
		IF eStatOld <> TLBuzActIdle
			AND eStatOld <> TLBuzActSetGreen
			AND eStatOld <> TLBuzActSetAmber
			AND eStatOld <> TLBuzActSetRed
			AND eStatOld <> TLBuzActSetBlue
			AND eStatOld <> TLBuzActSetWhite
			AND eStatOld <> TLBuzActSetBuz
			AND eStatOld <> TLBuzActRstGreen
			AND eStatOld <> TLBuzActRstAmber
			AND eStatOld <> TLBuzActRstRed
			AND eStatOld <> TLBuzActRstBlue
			AND eStatOld <> TLBuzActRstWhite
			AND eStatOld <> TLBuzActRstBuz
			AND eStatOld <> TLBuzActSetAll
			AND eStatOld <> TLBuzActRstAll THEN

			tylocalTLBuz.Out.bTLGreen	:= FALSE;
			tylocalTLBuz.Out.bTLAmber	:= FALSE;
			tylocalTLBuz.Out.bTLWhite	:= FALSE;
			tylocalTLBuz.Out.bTLBlue		:= FALSE;
			tylocalTLBuz.Out.bTLRed		:= FALSE;
			tylocalTLBuz.Out.bBuzBeep	:= FALSE;

		END_IF

		tylocalTLBuz.Out.sStatTxt	:= a_sStatText[tylocalTLBuz.Out.eStat];

		eStatOld	:= tylocalTLBuz.Out.eStat;

		tylocalTLBuz.Out.eStatus		:= Busy;
	END_IF

	//Main
	CASE tylocalTLBuz.Out.eStat OF

		TLBuzActIdle:
			IF tylocalTLBuz.Out.eStatus <> Idle THEN	//Reset Data
				//Private

				tylocalTLBuz.Out.sStatTxt	:= a_sStatText[tylocalTLBuz.Out.eStat];

			END_IF

			tylocalTLBuz.Out.eStatus	:= Idle;

		TLBuzActSetGreen:
			IF tylocalTLBuz.Out.eStatus = Idle OR tylocalTLBuz.Out.eStatus = Busy THEN

				tylocalTLBuz.Out.sStatTxt	:= a_sStatText[tylocalTLBuz.Out.eStat];

				tylocalTLBuz.Out.bTLGreen	:= TRUE;
				tylocalTLBuz.Out.eStatus		:= Done;

			END_IF

		TLBuzActSetAmber:
			IF tylocalTLBuz.Out.eStatus = Idle OR tylocalTLBuz.Out.eStatus = Busy THEN

				tylocalTLBuz.Out.sStatTxt	:= a_sStatText[tylocalTLBuz.Out.eStat];

				tylocalTLBuz.Out.bTLAmber	:= TRUE;
				tylocalTLBuz.Out.eStatus		:= Done;

			END_IF

		TLBuzActSetRed:
			IF tylocalTLBuz.Out.eStatus = Idle OR tylocalTLBuz.Out.eStatus = Busy THEN

				tylocalTLBuz.Out.sStatTxt	:= a_sStatText[tylocalTLBuz.Out.eStat];

				tylocalTLBuz.Out.bTLRed	:= TRUE;
				tylocalTLBuz.Out.eStatus	:= Done;

			END_IF

		TLBuzActSetBlue:
			IF tylocalTLBuz.Out.eStatus = Idle OR tylocalTLBuz.Out.eStatus = Busy THEN

				tylocalTLBuz.Out.sStatTxt	:= a_sStatText[tylocalTLBuz.Out.eStat];

				tylocalTLBuz.Out.bTLBlue		:= TRUE;
				tylocalTLBuz.Out.eStatus		:= Done;

			END_IF

		TLBuzActSetWhite:
			IF tylocalTLBuz.Out.eStatus = Idle OR tylocalTLBuz.Out.eStatus = Busy THEN

				tylocalTLBuz.Out.sStatTxt	:= a_sStatText[tylocalTLBuz.Out.eStat];

				tylocalTLBuz.Out.bTLWhite	:= TRUE;
				tylocalTLBuz.Out.eStatus		:= Done;

			END_IF

		TLBuzActSetBuz:
			IF tylocalTLBuz.Out.eStatus = Idle OR tylocalTLBuz.Out.eStatus = Busy THEN

				tylocalTLBuz.Out.sStatTxt	:= a_sStatText[tylocalTLBuz.Out.eStat];

				tylocalTLBuz.Out.bBuzBeep	:= TRUE;
				tylocalTLBuz.Out.eStatus		:= Done;

			END_IF

		TLBuzActRstGreen:
			IF tylocalTLBuz.Out.eStatus = Idle OR tylocalTLBuz.Out.eStatus = Busy THEN

				tylocalTLBuz.Out.sStatTxt	:= a_sStatText[tylocalTLBuz.Out.eStat];

				tylocalTLBuz.Out.bTLGreen	:= FALSE;
				tylocalTLBuz.Out.eStatus		:= Done;

			END_IF

		TLBuzActRstAmber:
			IF tylocalTLBuz.Out.eStatus = Idle OR tylocalTLBuz.Out.eStatus = Busy THEN

				tylocalTLBuz.Out.sStatTxt	:= a_sStatText[tylocalTLBuz.Out.eStat];

				tylocalTLBuz.Out.bTLAmber	:= FALSE;
				tylocalTLBuz.Out.eStatus		:= Done;

			END_IF

		TLBuzActRstRed:
			IF tylocalTLBuz.Out.eStatus = Idle OR tylocalTLBuz.Out.eStatus = Busy THEN

				tylocalTLBuz.Out.sStatTxt	:= a_sStatText[tylocalTLBuz.Out.eStat];

				tylocalTLBuz.Out.bTLRed		:= FALSE;
				tylocalTLBuz.Out.eStatus		:= Done;

			END_IF

		TLBuzActRstBlue:
			IF tylocalTLBuz.Out.eStatus = Idle OR tylocalTLBuz.Out.eStatus = Busy THEN

				tylocalTLBuz.Out.sStatTxt	:= a_sStatText[tylocalTLBuz.Out.eStat];

				tylocalTLBuz.Out.bTLBlue		:= FALSE;
				tylocalTLBuz.Out.eStatus		:= Done;

			END_IF

		TLBuzActRstWhite:
			IF tylocalTLBuz.Out.eStatus = Idle OR tylocalTLBuz.Out.eStatus = Busy THEN

				tylocalTLBuz.Out.sStatTxt	:= a_sStatText[tylocalTLBuz.Out.eStat];

				tylocalTLBuz.Out.bTLWhite	:= FALSE;
				tylocalTLBuz.Out.eStatus		:= Done;

			END_IF

		TLBuzActRstBuz:
			IF tylocalTLBuz.Out.eStatus = Idle OR tylocalTLBuz.Out.eStatus = Busy THEN

				tylocalTLBuz.Out.sStatTxt	:= a_sStatText[tylocalTLBuz.Out.eStat];

				tylocalTLBuz.Out.bBuzBeep	:= FALSE;
				tylocalTLBuz.Out.eStatus		:= Done;

			END_IF

		TLBuzActSetAll:
			IF tylocalTLBuz.Out.eStatus = Idle OR tylocalTLBuz.Out.eStatus = Busy THEN

				tylocalTLBuz.Out.sStatTxt	:= a_sStatText[tylocalTLBuz.Out.eStat];

				tylocalTLBuz.Out.bTLGreen	:= TRUE;
				tylocalTLBuz.Out.bTLRed		:= TRUE;
				tylocalTLBuz.Out.bTLAmber	:= TRUE;
				tylocalTLBuz.Out.bTLWhite	:= TRUE;
				tylocalTLBuz.Out.bTLBlue		:= TRUE;
				tylocalTLBuz.Out.bBuzBeep	:= TRUE;
				tylocalTLBuz.Out.eStatus		:= Done;

			END_IF

		TLBuzActRstAll:
			IF tylocalTLBuz.Out.eStatus = Idle OR tylocalTLBuz.Out.eStatus = Busy THEN

				tylocalTLBuz.Out.sStatTxt	:= a_sStatText[tylocalTLBuz.Out.eStat];

				tylocalTLBuz.Out.bTLGreen	:= FALSE;
				tylocalTLBuz.Out.bTLAmber	:= FALSE;
				tylocalTLBuz.Out.bTLRed		:= FALSE;
				tylocalTLBuz.Out.bTLWhite	:= FALSE;
				tylocalTLBuz.Out.bTLBlue		:= FALSE;
				tylocalTLBuz.Out.bBuzBeep	:= FALSE;
				tylocalTLBuz.Out.eStatus		:= Done;

			END_IF

	END_CASE

END_ACTION
```

#### Act_Background.st - Do Not Change!!!
```iecst
ACTION Act_Background: //For Standard Machines

	IF EDGEPOS(tylocalTLBuz.In.bUIManualMod) THEN

		fbBlink(bEn := FALSE);
		fbWarning(bEn := FALSE);

		tylocalTLBuz.Out.bTLRed		:= FALSE;
		tylocalTLBuz.Out.bTLAmber	:= TRUE;
		tylocalTLBuz.Out.bTLGreen	:= FALSE;
		tylocalTLBuz.Out.bBuzBeep	:= FALSE;

	ELSIF tylocalTLBuz.In.bUIManualMod THEN

		IF tylocalTLBuz.In.bErr = TRUE THEN

			fbBlink.tOnTm	:= tylocalTLBuz.In.tTLErrBlinkTm; //Error T#500ms (from NtParam)
			fbBlink.tOffTm	:= tylocalTLBuz.In.tTLErrBlinkTm; //Error T#500ms (from NtParam)

			fbWarning.tOnTm					:= tylocalTLBuz.In.tBuzErrOnTm; //Warn T#500ms (from NtParam)
			fbWarning.tOffTm				:= tylocalTLBuz.In.tBuzErrOnTm; //Warn T#500ms (from NtParam)
			fbWarning.tRstTm				:= tylocalTLBuz.In.tBuzErrRestTm; //Rest 5 seconds (from NtParam)
			fbWarning.usiOnCnt				:= tylocalTLBuz.In.usiBuzErrOnCntr; //Count 3 times (from NtParam)
			fbWarning.bStopAftRptSeqEn		:= tylocalTLBuz.In.bBuzErrStopSeqEn; //Enable Sequence Count (from NtParam)
			fbWarning.usiStopAftRptSeqCntr	:= tylocalTLBuz.In.usiBuzErrStopSeqCntr; //Sequence Counter  (from NtParam)

			fbBlink(bEn := TRUE);
			fbWarning(bEn := TRUE);

			tylocalTLBuz.Out.bTLRed		:= fbBlink.bOut;
			tylocalTLBuz.Out.bBuzBeep	:= (fbWarning.bOut) AND (tylocalTLBuz.In.bMuteBuz = FALSE);

			bManualErrOn := TRUE;

		ELSIF bManualErrOn THEN

			fbBlink(bEn := FALSE);
			fbWarning(bEn := FALSE);

			tylocalTLBuz.Out.bTLRed		:= FALSE;
			tylocalTLBuz.Out.bBuzBeep	:= FALSE;

			bManualErrOn := FALSE;

		END_IF

	ELSIF tylocalTLBuz.In.bUIManualMod = FALSE THEN

		bManualErrOn := FALSE;

		IF tylocalTLBuz.In.bStartup = TRUE THEN

			fbBlink(bEn := FALSE);
			fbWarning(bEn := FALSE);

			tylocalTLBuz.Out.bTLRed		:= TRUE;
			tylocalTLBuz.Out.bTLAmber	:= TRUE;
			tylocalTLBuz.Out.bTLGreen	:= TRUE;
			tylocalTLBuz.Out.bBuzBeep	:= FALSE;

		ELSIF tylocalTLBuz.In.bErr = TRUE THEN

			fbBlink.tOnTm	:= tylocalTLBuz.In.tTLErrBlinkTm; //Error T#500ms (from NtParam)
			fbBlink.tOffTm	:= tylocalTLBuz.In.tTLErrBlinkTm; //Error T#500ms (from NtParam)

			fbWarning.tOnTm					:= tylocalTLBuz.In.tBuzErrOnTm; //Warn T#500ms (from NtParam)
			fbWarning.tOffTm				:= tylocalTLBuz.In.tBuzErrOnTm; //Warn T#500ms (from NtParam)
			fbWarning.tRstTm				:= tylocalTLBuz.In.tBuzErrRestTm; //Rest 5 seconds (from NtParam)
			fbWarning.usiOnCnt				:= tylocalTLBuz.In.usiBuzErrOnCntr; //Count 3 times (from NtParam)
			fbWarning.bStopAftRptSeqEn		:= tylocalTLBuz.In.bBuzErrStopSeqEn; //Enable Sequence Count (from NtParam)
			fbWarning.usiStopAftRptSeqCntr	:= tylocalTLBuz.In.usiBuzErrStopSeqCntr; //Sequence Counter  (from NtParam)

			fbBlink(bEn := TRUE);
			fbWarning(bEn := TRUE);

			tylocalTLBuz.Out.bTLRed		:= fbBlink.bOut;
			tylocalTLBuz.Out.bTLAmber	:= FALSE;
			tylocalTLBuz.Out.bTLGreen	:= FALSE;
			tylocalTLBuz.Out.bBuzBeep	:= (fbWarning.bOut) AND (tylocalTLBuz.In.bMuteBuz = FALSE);

		ELSIF tylocalTLBuz.In.bErrNoBuz = TRUE THEN

			fbBlink.tOnTm	:= tylocalTLBuz.In.tTLErrBlinkTm;
			fbBlink.tOffTm	:= tylocalTLBuz.In.tTLErrBlinkTm;
			fbBlink(bEn := TRUE);
			fbWarning(bEn := FALSE);

			tylocalTLBuz.Out.bTLRed		:= fbBlink.bOut;
			tylocalTLBuz.Out.bTLAmber	:= FALSE;
			tylocalTLBuz.Out.bTLGreen	:= FALSE;
			tylocalTLBuz.Out.bBuzBeep	:= FALSE;

		ELSIF tylocalTLBuz.In.bWarning[0] = TRUE THEN

			fbBlink.tOnTm	:= tylocalTLBuz.In.tTLWarnBlinkTm[0]; //Warn T#500ms (from NtParam)
			fbBlink.tOffTm	:= tylocalTLBuz.In.tTLWarnBlinkTm[0]; //Warn T#500ms (from NtParam)

			fbWarning.tOnTm					:= tylocalTLBuz.In.tBuzWarnOnTm[0]; //Warn T#500ms (from NtParam)
			fbWarning.tOffTm				:= tylocalTLBuz.In.tBuzWarnOnTm[0]; //Warn T#500ms (from NtParam)
			fbWarning.tRstTm				:= tylocalTLBuz.In.tBuzWarnRestTm[0]; //Rest 5 seconds (from NtParam)
			fbWarning.usiOnCnt				:= tylocalTLBuz.In.usiBuzWarnOnCntr[0]; //Count 3 times (from NtParam)
			fbWarning.bStopAftRptSeqEn		:= tylocalTLBuz.In.bBuzWarnStopSeqEn[0]; //Enable Sequence Count (from NtParam)
			fbWarning.usiStopAftRptSeqCntr	:= tylocalTLBuz.In.usiBuzWarnStopSeqCntr[0]; //Sequence Counter  (from NtParam)

			fbBlink(bEn := TRUE);
			fbWarning(bEn := TRUE);

			tylocalTLBuz.Out.bTLRed		:= tylocalTLBuz.In.bStandby;
			tylocalTLBuz.Out.bTLAmber	:= fbBlink.bOut;
			tylocalTLBuz.Out.bTLGreen	:= tylocalTLBuz.In.bOps;
			tylocalTLBuz.Out.bBuzBeep	:= fbWarning.bOut AND (tylocalTLBuz.In.bMuteBuz = FALSE);

		ELSIF tylocalTLBuz.In.bWarningNoBuz[0] = TRUE THEN

			fbBlink.tOnTm	:= tylocalTLBuz.In.tTLWarnBlinkTm[0];
			fbBlink.tOffTm	:= tylocalTLBuz.In.tTLWarnBlinkTm[0];
			fbBlink(bEn := TRUE);
			fbWarning(bEn := FALSE);

			tylocalTLBuz.Out.bTLRed		:= tylocalTLBuz.In.bStandby;
			tylocalTLBuz.Out.bTLAmber	:= fbBlink.bOut;
			tylocalTLBuz.Out.bTLGreen	:= tylocalTLBuz.In.bOps;
			tylocalTLBuz.Out.bBuzBeep	:= FALSE;

		ELSIF tylocalTLBuz.In.bWarning[1] = TRUE THEN

			fbBlink.tOnTm	:= tylocalTLBuz.In.tTLWarnBlinkTm[1];
			fbBlink.tOffTm	:= tylocalTLBuz.In.tTLWarnBlinkTm[1];

			fbWarning.tOnTm					:= tylocalTLBuz.In.tBuzWarnOnTm[1]; //Warn T#500ms (from NtParam)
			fbWarning.tOffTm				:= tylocalTLBuz.In.tBuzWarnOnTm[1]; //Warn T#500ms (from NtParam)
			fbWarning.tRstTm				:= tylocalTLBuz.In.tBuzWarnRestTm[1]; //Rest 5 seconds (from NtParam)
			fbWarning.usiOnCnt				:= tylocalTLBuz.In.usiBuzWarnOnCntr[1]; //Count 3 times (from NtParam)
			fbWarning.bStopAftRptSeqEn		:= tylocalTLBuz.In.bBuzWarnStopSeqEn[1]; //Enable Sequence Count (from NtParam)
			fbWarning.usiStopAftRptSeqCntr	:= tylocalTLBuz.In.usiBuzWarnStopSeqCntr[1]; //Sequence Counter  (from NtParam)

			fbBlink(bEn := TRUE);
			fbWarning(bEn := TRUE);

			tylocalTLBuz.Out.bTLRed		:= tylocalTLBuz.In.bStandby;
			tylocalTLBuz.Out.bTLAmber	:= fbBlink.bOut;
			tylocalTLBuz.Out.bTLGreen	:= tylocalTLBuz.In.bOps;
			tylocalTLBuz.Out.bBuzBeep	:= fbWarning.bOut AND (tylocalTLBuz.In.bMuteBuz = FALSE);

		ELSIF tylocalTLBuz.In.bWarningNoBuz[1] = TRUE THEN

			fbBlink.tOnTm	:= tylocalTLBuz.In.tTLWarnBlinkTm[1];
			fbBlink.tOffTm	:= tylocalTLBuz.In.tTLWarnBlinkTm[1];
			fbBlink(bEn := TRUE);
			fbWarning(bEn := FALSE);

			tylocalTLBuz.Out.bTLRed		:= tylocalTLBuz.In.bStandby;
			tylocalTLBuz.Out.bTLAmber	:= fbBlink.bOut;
			tylocalTLBuz.Out.bTLGreen	:= tylocalTLBuz.In.bOps;
			tylocalTLBuz.Out.bBuzBeep	:= FALSE;

		ELSIF tylocalTLBuz.In.bWarning[2] = TRUE THEN

			fbBlink.tOnTm	:= tylocalTLBuz.In.tTLWarnBlinkTm[2];
			fbBlink.tOffTm	:= tylocalTLBuz.In.tTLWarnBlinkTm[2];

			fbWarning.tOnTm					:= tylocalTLBuz.In.tBuzWarnOnTm[2]; //Warn T#500ms (from NtParam)
			fbWarning.tOffTm				:= tylocalTLBuz.In.tBuzWarnOnTm[2]; //Warn T#500ms (from NtParam)
			fbWarning.tRstTm				:= tylocalTLBuz.In.tBuzWarnRestTm[2]; //Rest 5 seconds (from NtParam)
			fbWarning.usiOnCnt				:= tylocalTLBuz.In.usiBuzWarnOnCntr[2]; //Count 3 times (from NtParam)
			fbWarning.bStopAftRptSeqEn		:= tylocalTLBuz.In.bBuzWarnStopSeqEn[2]; //Enable Sequence Count (from NtParam)
			fbWarning.usiStopAftRptSeqCntr	:= tylocalTLBuz.In.usiBuzWarnStopSeqCntr[2]; //Sequence Counter  (from NtParam)

			fbBlink(bEn := TRUE);
			fbWarning(bEn := TRUE);

			tylocalTLBuz.Out.bTLRed		:= tylocalTLBuz.In.bStandby;
			tylocalTLBuz.Out.bTLAmber	:= fbBlink.bOut;
			tylocalTLBuz.Out.bTLGreen	:= tylocalTLBuz.In.bOps;
			tylocalTLBuz.Out.bBuzBeep	:= fbWarning.bOut AND (tylocalTLBuz.In.bMuteBuz = FALSE);

		ELSIF tylocalTLBuz.In.bWarningNoBuz[2] = TRUE THEN

			fbBlink.tOnTm	:= tylocalTLBuz.In.tTLWarnBlinkTm[2];
			fbBlink.tOffTm	:= tylocalTLBuz.In.tTLWarnBlinkTm[2];
			fbBlink(bEn := TRUE);
			fbWarning(bEn := FALSE);

			tylocalTLBuz.Out.bTLRed		:= tylocalTLBuz.In.bStandby;
			tylocalTLBuz.Out.bTLAmber	:= fbBlink.bOut;
			tylocalTLBuz.Out.bTLGreen	:= tylocalTLBuz.In.bOps;
			tylocalTLBuz.Out.bBuzBeep	:= FALSE;

		ELSIF tylocalTLBuz.In.bWarning[3] = TRUE THEN

			fbBlink.tOnTm	:= tylocalTLBuz.In.tTLWarnBlinkTm[3];
			fbBlink.tOffTm	:= tylocalTLBuz.In.tTLWarnBlinkTm[3];

			fbWarning.tOnTm					:= tylocalTLBuz.In.tBuzWarnOnTm[3]; //Warn T#500ms (from NtParam)
			fbWarning.tOffTm				:= tylocalTLBuz.In.tBuzWarnOnTm[3]; //Warn T#500ms (from NtParam)
			fbWarning.tRstTm				:= tylocalTLBuz.In.tBuzWarnRestTm[3]; //Rest 5 seconds (from NtParam)
			fbWarning.usiOnCnt				:= tylocalTLBuz.In.usiBuzWarnOnCntr[3]; //Count 3 times (from NtParam)
			fbWarning.bStopAftRptSeqEn		:= tylocalTLBuz.In.bBuzWarnStopSeqEn[3]; //Enable Sequence Count (from NtParam)
			fbWarning.usiStopAftRptSeqCntr	:= tylocalTLBuz.In.usiBuzWarnStopSeqCntr[3]; //Sequence Counter  (from NtParam)

			fbBlink(bEn := TRUE);
			fbWarning(bEn := TRUE);

			tylocalTLBuz.Out.bTLRed		:= tylocalTLBuz.In.bStandby;
			tylocalTLBuz.Out.bTLAmber	:= fbBlink.bOut;
			tylocalTLBuz.Out.bTLGreen	:= tylocalTLBuz.In.bOps;
			tylocalTLBuz.Out.bBuzBeep	:= fbWarning.bOut AND (tylocalTLBuz.In.bMuteBuz = FALSE);

		ELSIF tylocalTLBuz.In.bWarningNoBuz[3] = TRUE THEN

			fbBlink.tOnTm	:= tylocalTLBuz.In.tTLWarnBlinkTm[3];
			fbBlink.tOffTm	:= tylocalTLBuz.In.tTLWarnBlinkTm[3];
			fbBlink(bEn := TRUE);
			fbWarning(bEn := FALSE);

			tylocalTLBuz.Out.bTLRed		:= tylocalTLBuz.In.bStandby;
			tylocalTLBuz.Out.bTLAmber	:= fbBlink.bOut;
			tylocalTLBuz.Out.bTLGreen	:= tylocalTLBuz.In.bOps;
			tylocalTLBuz.Out.bBuzBeep	:= FALSE;

		ELSIF tylocalTLBuz.In.bWarning[4] = TRUE THEN

			fbBlink.tOnTm	:= tylocalTLBuz.In.tTLWarnBlinkTm[4];
			fbBlink.tOffTm	:= tylocalTLBuz.In.tTLWarnBlinkTm[4];

			fbWarning.tOnTm					:= tylocalTLBuz.In.tBuzWarnOnTm[4]; //Warn T#500ms (from NtParam)
			fbWarning.tOffTm				:= tylocalTLBuz.In.tBuzWarnOnTm[4]; //Warn T#500ms (from NtParam)
			fbWarning.tRstTm				:= tylocalTLBuz.In.tBuzWarnRestTm[4]; //Rest 5 seconds (from NtParam)
			fbWarning.usiOnCnt				:= tylocalTLBuz.In.usiBuzWarnOnCntr[4]; //Count 3 times (from NtParam)
			fbWarning.bStopAftRptSeqEn		:= tylocalTLBuz.In.bBuzWarnStopSeqEn[4]; //Enable Sequence Count (from NtParam)
			fbWarning.usiStopAftRptSeqCntr	:= tylocalTLBuz.In.usiBuzWarnStopSeqCntr[4]; //Sequence Counter  (from NtParam)

			fbBlink(bEn := TRUE);
			fbWarning(bEn := TRUE);

			tylocalTLBuz.Out.bTLRed		:= tylocalTLBuz.In.bStandby;
			tylocalTLBuz.Out.bTLAmber	:= fbBlink.bOut;
			tylocalTLBuz.Out.bTLGreen	:= tylocalTLBuz.In.bOps;
			tylocalTLBuz.Out.bBuzBeep	:= fbWarning.bOut AND (tylocalTLBuz.In.bMuteBuz = FALSE);

		ELSIF tylocalTLBuz.In.bWarningNoBuz[4] = TRUE THEN

			fbBlink.tOnTm	:= tylocalTLBuz.In.tTLWarnBlinkTm[4];
			fbBlink.tOffTm	:= tylocalTLBuz.In.tTLWarnBlinkTm[4];
			fbBlink(bEn := TRUE);
			fbWarning(bEn := FALSE);

			tylocalTLBuz.Out.bTLRed		:= tylocalTLBuz.In.bStandby;
			tylocalTLBuz.Out.bTLAmber	:= fbBlink.bOut;
			tylocalTLBuz.Out.bTLGreen	:= tylocalTLBuz.In.bOps;
			tylocalTLBuz.Out.bBuzBeep	:= FALSE;

		ELSIF tylocalTLBuz.In.bWarning[5] = TRUE THEN

			fbBlink.tOnTm	:= tylocalTLBuz.In.tTLWarnBlinkTm[5];
			fbBlink.tOffTm	:= tylocalTLBuz.In.tTLWarnBlinkTm[5];

			fbWarning.tOnTm					:= tylocalTLBuz.In.tBuzWarnOnTm[5]; //Warn T#500ms (from NtParam)
			fbWarning.tOffTm				:= tylocalTLBuz.In.tBuzWarnOnTm[5]; //Warn T#500ms (from NtParam)
			fbWarning.tRstTm				:= tylocalTLBuz.In.tBuzWarnRestTm[5]; //Rest 5 seconds (from NtParam)
			fbWarning.usiOnCnt				:= tylocalTLBuz.In.usiBuzWarnOnCntr[5]; //Count 3 times (from NtParam)
			fbWarning.bStopAftRptSeqEn		:= tylocalTLBuz.In.bBuzWarnStopSeqEn[5]; //Enable Sequence Count (from NtParam)
			fbWarning.usiStopAftRptSeqCntr	:= tylocalTLBuz.In.usiBuzWarnStopSeqCntr[5]; //Sequence Counter  (from NtParam)

			fbBlink(bEn := TRUE);
			fbWarning(bEn := TRUE);

			tylocalTLBuz.Out.bTLRed		:= tylocalTLBuz.In.bStandby;
			tylocalTLBuz.Out.bTLAmber	:= fbBlink.bOut;
			tylocalTLBuz.Out.bTLGreen	:= tylocalTLBuz.In.bOps;
			tylocalTLBuz.Out.bBuzBeep	:= fbWarning.bOut AND (tylocalTLBuz.In.bMuteBuz = FALSE);

		ELSIF tylocalTLBuz.In.bWarningNoBuz[5] = TRUE THEN

			fbBlink.tOnTm	:= tylocalTLBuz.In.tTLWarnBlinkTm[5];
			fbBlink.tOffTm	:= tylocalTLBuz.In.tTLWarnBlinkTm[5];
			fbBlink(bEn := TRUE);
			fbWarning(bEn := FALSE);

			tylocalTLBuz.Out.bTLRed		:= tylocalTLBuz.In.bStandby;
			tylocalTLBuz.Out.bTLAmber	:= fbBlink.bOut;
			tylocalTLBuz.Out.bTLGreen	:= tylocalTLBuz.In.bOps;
			tylocalTLBuz.Out.bBuzBeep	:= FALSE;

		ELSIF tylocalTLBuz.In.bSeqStop = TRUE THEN

			fbBlink.tOnTm	:= tBlinkTm;
			fbBlink.tOffTm	:= tBlinkTm;
			fbBlink(bEn := TRUE);
			fbWarning(bEn := FALSE);

			tylocalTLBuz.Out.bTLRed		:= fbBlink.bOut;
			tylocalTLBuz.Out.bTLAmber	:= FALSE;
			tylocalTLBuz.Out.bTLGreen	:= TRUE;
			tylocalTLBuz.Out.bBuzBeep	:= FALSE;

		ELSIF tylocalTLBuz.In.bChgRcp = TRUE THEN

			fbBlink.tOnTm	:= tylocalTLBuz.In.tTLChgRcpBlinkTm;
			fbBlink.tOffTm	:= tylocalTLBuz.In.tTLChgRcpBlinkTm;
			fbBlink(bEn := TRUE);
			fbWarning(bEn := FALSE);

			IF EDGE(fbBlink.bOut) THEN
				IF tylocalTLBuz.Out.bTLRed = TRUE THEN
					tylocalTLBuz.Out.bTLRed		:= FALSE;
					tylocalTLBuz.Out.bTLAmber	:= FALSE;
					tylocalTLBuz.Out.bTLGreen	:= TRUE;
				ELSIF tylocalTLBuz.Out.bTLAmber = TRUE THEN
					tylocalTLBuz.Out.bTLRed		:= TRUE;
					tylocalTLBuz.Out.bTLAmber	:= FALSE;
					tylocalTLBuz.Out.bTLGreen	:= FALSE;
				ELSE
					tylocalTLBuz.Out.bTLRed		:= FALSE;
					tylocalTLBuz.Out.bTLAmber	:= TRUE;
					tylocalTLBuz.Out.bTLGreen	:= FALSE;
				END_IF
			END_IF

			tylocalTLBuz.Out.bBuzBeep	:= fbBlink.bOut AND (tylocalTLBuz.In.bMuteBuz = FALSE);

		ELSIF tylocalTLBuz.In.bStep = TRUE THEN

			fbBlink.tOnTm	:= tBlinkTm;
			fbBlink.tOffTm	:= tBlinkTm;
			fbBlink(bEn := TRUE);
			fbWarning(bEn := FALSE);

			tylocalTLBuz.Out.bTLRed		:= FALSE;
			tylocalTLBuz.Out.bTLAmber	:= FALSE;
			tylocalTLBuz.Out.bTLGreen	:= fbBlink.bOut;
			tylocalTLBuz.Out.bBuzBeep	:= FALSE;

		ELSIF tylocalTLBuz.In.bOps = TRUE THEN

			fbBlink(bEn := FALSE);
			fbWarning(bEn := FALSE);

			tylocalTLBuz.Out.bTLRed		:= FALSE;
			tylocalTLBuz.Out.bTLAmber	:= FALSE;
			tylocalTLBuz.Out.bTLGreen	:= TRUE;
			tylocalTLBuz.Out.bBuzBeep	:= FALSE;

		ELSIF tylocalTLBuz.In.bSimulation = TRUE THEN

			fbBlink.tOnTm	:= tBlinkTm;
			fbBlink.tOffTm	:= tBlinkTm;
			fbBlink(bEn := TRUE);
			fbWarning(bEn := FALSE);

			tylocalTLBuz.Out.bTLRed		:= fbBlink.bOut;
			tylocalTLBuz.Out.bTLAmber	:= fbBlink.bOut;
			tylocalTLBuz.Out.bTLGreen	:= TRUE;
			tylocalTLBuz.Out.bBuzBeep	:= FALSE;

		ELSIF tylocalTLBuz.In.bStandby = TRUE THEN

			fbBlink(bEn := FALSE);
			fbWarning(bEn := FALSE);

			tylocalTLBuz.Out.bTLRed		:= TRUE;
			tylocalTLBuz.Out.bTLAmber	:= FALSE;
			tylocalTLBuz.Out.bTLGreen	:= FALSE;
			tylocalTLBuz.Out.bBuzBeep	:= FALSE;

		ELSE

			fbBlink(bEn := FALSE);
			fbWarning(bEn := FALSE);

			tylocalTLBuz.Out.bTLRed		:= FALSE;
			tylocalTLBuz.Out.bTLAmber	:= FALSE;
			tylocalTLBuz.Out.bTLGreen	:= FALSE;
			tylocalTLBuz.Out.bBuzBeep	:= FALSE;

		END_IF

	END_IF

	IF tylocalTLBuz.In.bUIManualMod = FALSE AND tylocalTLBuz.In.bErr = FALSE THEN
		IF tylocalTLBuz.In.bTLAmberFlashEn THEN //Amber Flash 1 sec [Put Conditions in Act_Link.st]

			fbBlink1.tOnTm	:= tylocalTLBuz.In.tTLAmberBlinkTm; //T#500ms (from NtParam)
			fbBlink1.tOffTm	:= tylocalTLBuz.In.tTLAmberBlinkTm; //T#500ms (from NtParam)
			fbBlink1(bEn := TRUE);

			tylocalTLBuz.Out.bTLAmber	:= fbBlink1.bOut;

		ELSE
			fbBlink1(bEn := FALSE);
		END_IF

		IF tylocalTLBuz.In.bTLRedFlashEn THEN //Red Flash 1 sec [Put Conditions in Act_Link.st]

			fbBlink2.tOnTm	:= tylocalTLBuz.In.tTLRedBlinkTm; //T#500ms (from NtParam)
			fbBlink2.tOffTm	:= tylocalTLBuz.In.tTLRedBlinkTm; //T#500ms (from NtParam)
			fbBlink2(bEn := TRUE);

			tylocalTLBuz.Out.bTLRed		:= fbBlink2.bOut;
		ELSE
			fbBlink2(bEn := FALSE);
		END_IF

		IF tylocalTLBuz.In.bTLGreenFlashEn THEN //Green Flash 1 sec [Put Conditions in Act_Link.st]

			fbBlink3.tOnTm	:= tylocalTLBuz.In.tTLGreenBlinkTm; //T#500ms (from NtParam)
			fbBlink3.tOffTm	:= tylocalTLBuz.In.tTLGreenBlinkTm; //T#500ms (from NtParam)
			fbBlink3(bEn := TRUE);

			tylocalTLBuz.Out.bTLGreen	:= fbBlink3.bOut;
		ELSE
			fbBlink3(bEn := FALSE);
		END_IF

		IF tylocalTLBuz.In.bBuzAlertEn = TRUE AND fbWarning.bEn=FALSE THEN

			fbWarning1.tOnTm				:= tylocalTLBuz.In.tBuzAlertOnTm;
			fbWarning1.tOffTm				:= tylocalTLBuz.In.tBuzAlertOnTm;
			fbWarning1.tRstTm				:= tylocalTLBuz.In.tBuzAlertRestTm;
			fbWarning1.usiOnCnt				:= tylocalTLBuz.In.usiBuzAlertOnCntr;
			fbWarning1.bStopAftRptSeqEn		:= tylocalTLBuz.In.bBuzAlertStopSeqEn; //Enable Sequence Count (from NtParam)
			fbWarning1.usiStopAftRptSeqCntr	:= tylocalTLBuz.In.usiBuzAlertStopSeqCntr; //Sequence Counter  (from NtParam)

			fbWarning1(bEn := TRUE);

			tylocalTLBuz.Out.bBuzBeep	:= fbWarning1.bOut AND (tylocalTLBuz.In.bMuteBuz = FALSE);

		ELSE
			fbWarning1(bEn := FALSE);
		END_IF
	ELSE
		fbBlink1(bEn := FALSE);
		fbBlink2(bEn := FALSE);
		fbBlink3(bEn := FALSE);
		fbWarning1(bEn := FALSE);
	END_IF

	//Arrange tylocalTLBuz.In.bWarning according to the severity of the warning or info (Err is prioritized)
	IF tylocalTLBuz.In.bErr THEN
		usiWarnInfoStateNew	:= 1;
	ELSIF tylocalTLBuz.In.bWarning[0] THEN
		usiWarnInfoStateNew	:= 2;
	ELSIF tylocalTLBuz.In.bWarning[1] THEN
		usiWarnInfoStateNew	:= 3;
	ELSIF tylocalTLBuz.In.bWarning[2] THEN
		usiWarnInfoStateNew	:= 4;
	ELSIF tylocalTLBuz.In.bWarning[3] THEN
		usiWarnInfoStateNew	:= 5;
	ELSIF tylocalTLBuz.In.bWarning[4] THEN
		usiWarnInfoStateNew	:= 6;
	ELSIF tylocalTLBuz.In.bWarning[5] THEN
		usiWarnInfoStateNew	:= 7;
	ELSIF tylocalTLBuz.In.bBuzAlertEn AND fbWarning.bEn=FALSE THEN
		usiWarnInfoStateNew	:= 8;
	ELSE
		usiWarnInfoStateNew	:= 0;
	END_IF

	IF usiWarnInfoStateOld<>usiWarnInfoStateNew THEN
		usiWarnInfoStateOld:=usiWarnInfoStateNew;
		fbWarning(bEn := FALSE);
		fbWarning1(bEn := FALSE);
	END_IF

END_ACTION
```

#### Act_Background1.st - Do Not Change!!!
```iecst
ACTION Act_Background1: //For Aptiv Machines

	IF EDGEPOS(tylocalTLBuz.In.bUIManualMod) THEN

		fbBlink(bEn := FALSE);
		fbWarning(bEn := FALSE);

		tylocalTLBuz.Out.bTLRed		:= FALSE;
		tylocalTLBuz.Out.bTLAmber	:= TRUE;
		tylocalTLBuz.Out.bTLGreen	:= FALSE;
		tylocalTLBuz.Out.bBuzBeep	:= FALSE;

	ELSIF tylocalTLBuz.In.bUIManualMod THEN

		IF tylocalTLBuz.In.bErr = TRUE THEN

			fbBlink.tOnTm	:= tylocalTLBuz.In.tTLErrBlinkTm; //Error T#500ms (from NtParam)
			fbBlink.tOffTm	:= tylocalTLBuz.In.tTLErrBlinkTm; //Error T#500ms (from NtParam)

			fbWarning.tOnTm					:= tylocalTLBuz.In.tBuzErrOnTm; //Warn T#500ms (from NtParam)
			fbWarning.tOffTm				:= tylocalTLBuz.In.tBuzErrOnTm; //Warn T#500ms (from NtParam)
			fbWarning.tRstTm				:= tylocalTLBuz.In.tBuzErrRestTm; //Rest 5 seconds (from NtParam)
			fbWarning.usiOnCnt				:= tylocalTLBuz.In.usiBuzErrOnCntr; //Count 3 times (from NtParam)
			fbWarning.bStopAftRptSeqEn		:= tylocalTLBuz.In.bBuzErrStopSeqEn; //Enable Sequence Count (from NtParam)
			fbWarning.usiStopAftRptSeqCntr	:= tylocalTLBuz.In.usiBuzErrStopSeqCntr; //Sequence Counter  (from NtParam)

			fbBlink(bEn := TRUE);
			fbWarning(bEn := TRUE);

			tylocalTLBuz.Out.bTLRed		:= TRUE;
			tylocalTLBuz.Out.bBuzBeep	:= (fbWarning.bOut) AND (tylocalTLBuz.In.bMuteBuz = FALSE);

			bManualErrOn := TRUE;

		ELSIF bManualErrOn THEN

			fbBlink(bEn := FALSE);
			fbWarning(bEn := FALSE);

			tylocalTLBuz.Out.bTLRed		:= FALSE;
			tylocalTLBuz.Out.bBuzBeep	:= FALSE;

			bManualErrOn := FALSE;

		END_IF

	ELSIF tylocalTLBuz.In.bUIManualMod = FALSE THEN

		bManualErrOn := FALSE;

		IF tylocalTLBuz.In.bStartup = TRUE THEN

			fbBlink(bEn := FALSE);
			fbWarning(bEn := FALSE);

			tylocalTLBuz.Out.bTLRed		:= TRUE;
			tylocalTLBuz.Out.bTLAmber	:= TRUE;
			tylocalTLBuz.Out.bTLGreen	:= TRUE;
			tylocalTLBuz.Out.bBuzBeep	:= FALSE;

		ELSIF tylocalTLBuz.In.bCoverSwitchSig = FALSE THEN

			fbBlink.tOnTm	:= tylocalTLBuz.In.tTLErrBlinkTm;
			fbBlink.tOffTm	:= tylocalTLBuz.In.tTLErrBlinkTm;
			fbBlink(bEn := TRUE);
			fbWarning(bEn := FALSE);

			tylocalTLBuz.Out.bTLRed		:= fbBlink.bOut;
			tylocalTLBuz.Out.bTLAmber	:= FALSE;
			tylocalTLBuz.Out.bTLGreen	:= FALSE;
			tylocalTLBuz.Out.bBuzBeep	:= (fbBlink.bOut) AND (tylocalTLBuz.In.bMuteBuz = FALSE);

		ELSIF tylocalTLBuz.In.bErr = TRUE THEN

			fbBlink.tOnTm	:= tylocalTLBuz.In.tTLErrBlinkTm; //Error T#500ms (from NtParam)
			fbBlink.tOffTm	:= tylocalTLBuz.In.tTLErrBlinkTm; //Error T#500ms (from NtParam)

			fbWarning.tOnTm					:= tylocalTLBuz.In.tBuzErrOnTm; //Warn T#500ms (from NtParam)
			fbWarning.tOffTm				:= tylocalTLBuz.In.tBuzErrOnTm; //Warn T#500ms (from NtParam)
			fbWarning.tRstTm				:= tylocalTLBuz.In.tBuzErrRestTm; //Rest 5 seconds (from NtParam)
			fbWarning.usiOnCnt				:= tylocalTLBuz.In.usiBuzErrOnCntr; //Count 3 times (from NtParam)
			fbWarning.bStopAftRptSeqEn		:= tylocalTLBuz.In.bBuzErrStopSeqEn; //Enable Sequence Count (from NtParam)
			fbWarning.usiStopAftRptSeqCntr	:= tylocalTLBuz.In.usiBuzErrStopSeqCntr; //Sequence Counter  (from NtParam)

			fbBlink(bEn := TRUE);
			fbWarning(bEn := TRUE);

			tylocalTLBuz.Out.bTLRed		:= TRUE;
			tylocalTLBuz.Out.bTLAmber	:= FALSE;
			tylocalTLBuz.Out.bTLGreen	:= FALSE;
			tylocalTLBuz.Out.bBuzBeep	:= (fbWarning.bOut) AND (tylocalTLBuz.In.bMuteBuz = FALSE);

		ELSIF tylocalTLBuz.In.bErrNoBuz = TRUE THEN

			fbBlink.tOnTm	:= tylocalTLBuz.In.tTLErrBlinkTm;
			fbBlink.tOffTm	:= tylocalTLBuz.In.tTLErrBlinkTm;
			fbBlink(bEn := TRUE);
			fbWarning(bEn := FALSE);

			tylocalTLBuz.Out.bTLRed		:= fbBlink.bOut;
			tylocalTLBuz.Out.bTLAmber	:= FALSE;
			tylocalTLBuz.Out.bTLGreen	:= FALSE;
			tylocalTLBuz.Out.bBuzBeep	:= FALSE;

		ELSIF tylocalTLBuz.In.bWarning[0] = TRUE THEN

			fbBlink.tOnTm	:= tylocalTLBuz.In.tTLWarnBlinkTm[0]; //Warn T#500ms (from NtParam)
			fbBlink.tOffTm	:= tylocalTLBuz.In.tTLWarnBlinkTm[0]; //Warn T#500ms (from NtParam)

			fbWarning.tOnTm					:= tylocalTLBuz.In.tBuzWarnOnTm[0]; //Warn T#500ms (from NtParam)
			fbWarning.tOffTm				:= tylocalTLBuz.In.tBuzWarnOnTm[0]; //Warn T#500ms (from NtParam)
			fbWarning.tRstTm				:= tylocalTLBuz.In.tBuzWarnRestTm[0]; //Rest 5 seconds (from NtParam)
			fbWarning.usiOnCnt				:= tylocalTLBuz.In.usiBuzWarnOnCntr[0]; //Count 3 times (from NtParam)
			fbWarning.bStopAftRptSeqEn		:= tylocalTLBuz.In.bBuzWarnStopSeqEn[0]; //Enable Sequence Count (from NtParam)
			fbWarning.usiStopAftRptSeqCntr	:= tylocalTLBuz.In.usiBuzWarnStopSeqCntr[0]; //Sequence Counter  (from NtParam)

			fbBlink(bEn := TRUE);
			fbWarning(bEn := TRUE);

			tylocalTLBuz.Out.bTLRed		:= FALSE;
			tylocalTLBuz.Out.bTLAmber	:= fbBlink.bOut;
			tylocalTLBuz.Out.bTLGreen	:= FALSE;
			tylocalTLBuz.Out.bBuzBeep	:= fbWarning.bOut AND (tylocalTLBuz.In.bMuteBuz = FALSE);

		ELSIF tylocalTLBuz.In.bWarningNoBuz[0] = TRUE THEN

			fbBlink.tOnTm	:= tylocalTLBuz.In.tTLWarnBlinkTm[0];
			fbBlink.tOffTm	:= tylocalTLBuz.In.tTLWarnBlinkTm[0];
			fbBlink(bEn := TRUE);
			fbWarning(bEn := FALSE);

			tylocalTLBuz.Out.bTLRed		:= FALSE;
			tylocalTLBuz.Out.bTLAmber	:= fbBlink.bOut;
			tylocalTLBuz.Out.bTLGreen	:= FALSE;
			tylocalTLBuz.Out.bBuzBeep	:= FALSE;

		ELSIF tylocalTLBuz.In.bWarning[1] = TRUE THEN

			fbBlink.tOnTm	:= tylocalTLBuz.In.tTLWarnBlinkTm[1];
			fbBlink.tOffTm	:= tylocalTLBuz.In.tTLWarnBlinkTm[1];

			fbWarning.tOnTm					:= tylocalTLBuz.In.tBuzWarnOnTm[1]; //Warn T#500ms (from NtParam)
			fbWarning.tOffTm				:= tylocalTLBuz.In.tBuzWarnOnTm[1]; //Warn T#500ms (from NtParam)
			fbWarning.tRstTm				:= tylocalTLBuz.In.tBuzWarnRestTm[1]; //Rest 5 seconds (from NtParam)
			fbWarning.usiOnCnt				:= tylocalTLBuz.In.usiBuzWarnOnCntr[1]; //Count 3 times (from NtParam)
			fbWarning.bStopAftRptSeqEn		:= tylocalTLBuz.In.bBuzWarnStopSeqEn[1]; //Enable Sequence Count (from NtParam)
			fbWarning.usiStopAftRptSeqCntr	:= tylocalTLBuz.In.usiBuzWarnStopSeqCntr[1]; //Sequence Counter  (from NtParam)

			fbBlink(bEn := TRUE);
			fbWarning(bEn := TRUE);

			tylocalTLBuz.Out.bTLRed		:= tylocalTLBuz.In.bStandby;
			tylocalTLBuz.Out.bTLAmber	:= fbBlink.bOut;
			tylocalTLBuz.Out.bTLGreen	:= tylocalTLBuz.In.bOps;
			tylocalTLBuz.Out.bBuzBeep	:= fbWarning.bOut AND (tylocalTLBuz.In.bMuteBuz = FALSE);

		ELSIF tylocalTLBuz.In.bWarningNoBuz[1] = TRUE THEN

			fbBlink.tOnTm	:= tylocalTLBuz.In.tTLWarnBlinkTm[1];
			fbBlink.tOffTm	:= tylocalTLBuz.In.tTLWarnBlinkTm[1];
			fbBlink(bEn := TRUE);
			fbWarning(bEn := FALSE);

			tylocalTLBuz.Out.bTLRed		:= tylocalTLBuz.In.bStandby;
			tylocalTLBuz.Out.bTLAmber	:= fbBlink.bOut;
			tylocalTLBuz.Out.bTLGreen	:= tylocalTLBuz.In.bOps;
			tylocalTLBuz.Out.bBuzBeep	:= FALSE;

		ELSIF tylocalTLBuz.In.bWarning[2] = TRUE THEN

			fbBlink.tOnTm	:= tylocalTLBuz.In.tTLWarnBlinkTm[2];
			fbBlink.tOffTm	:= tylocalTLBuz.In.tTLWarnBlinkTm[2];

			fbWarning.tOnTm					:= tylocalTLBuz.In.tBuzWarnOnTm[2]; //Warn T#500ms (from NtParam)
			fbWarning.tOffTm				:= tylocalTLBuz.In.tBuzWarnOnTm[2]; //Warn T#500ms (from NtParam)
			fbWarning.tRstTm				:= tylocalTLBuz.In.tBuzWarnRestTm[2]; //Rest 5 seconds (from NtParam)
			fbWarning.usiOnCnt				:= tylocalTLBuz.In.usiBuzWarnOnCntr[2]; //Count 3 times (from NtParam)
			fbWarning.bStopAftRptSeqEn		:= tylocalTLBuz.In.bBuzWarnStopSeqEn[2]; //Enable Sequence Count (from NtParam)
			fbWarning.usiStopAftRptSeqCntr	:= tylocalTLBuz.In.usiBuzWarnStopSeqCntr[2]; //Sequence Counter  (from NtParam)

			fbBlink(bEn := TRUE);
			fbWarning(bEn := TRUE);

			tylocalTLBuz.Out.bTLRed		:= tylocalTLBuz.In.bStandby;
			tylocalTLBuz.Out.bTLAmber	:= fbBlink.bOut;
			tylocalTLBuz.Out.bTLGreen	:= tylocalTLBuz.In.bOps;
			tylocalTLBuz.Out.bBuzBeep	:= fbWarning.bOut AND (tylocalTLBuz.In.bMuteBuz = FALSE);

		ELSIF tylocalTLBuz.In.bWarningNoBuz[2] = TRUE THEN

			fbBlink.tOnTm	:= tylocalTLBuz.In.tTLWarnBlinkTm[2];
			fbBlink.tOffTm	:= tylocalTLBuz.In.tTLWarnBlinkTm[2];
			fbBlink(bEn := TRUE);
			fbWarning(bEn := FALSE);

			tylocalTLBuz.Out.bTLRed		:= tylocalTLBuz.In.bStandby;
			tylocalTLBuz.Out.bTLAmber	:= fbBlink.bOut;
			tylocalTLBuz.Out.bTLGreen	:= tylocalTLBuz.In.bOps;
			tylocalTLBuz.Out.bBuzBeep	:= FALSE;

		ELSIF tylocalTLBuz.In.bWarning[3] = TRUE THEN

			fbBlink.tOnTm	:= tylocalTLBuz.In.tTLWarnBlinkTm[3];
			fbBlink.tOffTm	:= tylocalTLBuz.In.tTLWarnBlinkTm[3];

			fbWarning.tOnTm					:= tylocalTLBuz.In.tBuzWarnOnTm[3]; //Warn T#500ms (from NtParam)
			fbWarning.tOffTm				:= tylocalTLBuz.In.tBuzWarnOnTm[3]; //Warn T#500ms (from NtParam)
			fbWarning.tRstTm				:= tylocalTLBuz.In.tBuzWarnRestTm[3]; //Rest 5 seconds (from NtParam)
			fbWarning.usiOnCnt				:= tylocalTLBuz.In.usiBuzWarnOnCntr[3]; //Count 3 times (from NtParam)
			fbWarning.bStopAftRptSeqEn		:= tylocalTLBuz.In.bBuzWarnStopSeqEn[3]; //Enable Sequence Count (from NtParam)
			fbWarning.usiStopAftRptSeqCntr	:= tylocalTLBuz.In.usiBuzWarnStopSeqCntr[3]; //Sequence Counter  (from NtParam)

			fbBlink(bEn := TRUE);
			fbWarning(bEn := TRUE);

			tylocalTLBuz.Out.bTLRed		:= tylocalTLBuz.In.bStandby;
			tylocalTLBuz.Out.bTLAmber	:= fbBlink.bOut;
			tylocalTLBuz.Out.bTLGreen	:= tylocalTLBuz.In.bOps;
			tylocalTLBuz.Out.bBuzBeep	:= fbWarning.bOut AND (tylocalTLBuz.In.bMuteBuz = FALSE);

		ELSIF tylocalTLBuz.In.bWarningNoBuz[3] = TRUE THEN

			fbBlink.tOnTm	:= tylocalTLBuz.In.tTLWarnBlinkTm[3];
			fbBlink.tOffTm	:= tylocalTLBuz.In.tTLWarnBlinkTm[3];
			fbBlink(bEn := TRUE);
			fbWarning(bEn := FALSE);

			tylocalTLBuz.Out.bTLRed		:= tylocalTLBuz.In.bStandby;
			tylocalTLBuz.Out.bTLAmber	:= fbBlink.bOut;
			tylocalTLBuz.Out.bTLGreen	:= tylocalTLBuz.In.bOps;
			tylocalTLBuz.Out.bBuzBeep	:= FALSE;

		ELSIF tylocalTLBuz.In.bWarning[4] = TRUE THEN

			fbBlink.tOnTm	:= tylocalTLBuz.In.tTLWarnBlinkTm[4];
			fbBlink.tOffTm	:= tylocalTLBuz.In.tTLWarnBlinkTm[4];

			fbWarning.tOnTm					:= tylocalTLBuz.In.tBuzWarnOnTm[4]; //Warn T#500ms (from NtParam)
			fbWarning.tOffTm				:= tylocalTLBuz.In.tBuzWarnOnTm[4]; //Warn T#500ms (from NtParam)
			fbWarning.tRstTm				:= tylocalTLBuz.In.tBuzWarnRestTm[4]; //Rest 5 seconds (from NtParam)
			fbWarning.usiOnCnt				:= tylocalTLBuz.In.usiBuzWarnOnCntr[4]; //Count 3 times (from NtParam)
			fbWarning.bStopAftRptSeqEn		:= tylocalTLBuz.In.bBuzWarnStopSeqEn[4]; //Enable Sequence Count (from NtParam)
			fbWarning.usiStopAftRptSeqCntr	:= tylocalTLBuz.In.usiBuzWarnStopSeqCntr[4]; //Sequence Counter  (from NtParam)

			fbBlink(bEn := TRUE);
			fbWarning(bEn := TRUE);

			tylocalTLBuz.Out.bTLRed		:= tylocalTLBuz.In.bStandby;
			tylocalTLBuz.Out.bTLAmber	:= fbBlink.bOut;
			tylocalTLBuz.Out.bTLGreen	:= tylocalTLBuz.In.bOps;
			tylocalTLBuz.Out.bBuzBeep	:= fbWarning.bOut AND (tylocalTLBuz.In.bMuteBuz = FALSE);

		ELSIF tylocalTLBuz.In.bWarningNoBuz[4] = TRUE THEN

			fbBlink.tOnTm	:= tylocalTLBuz.In.tTLWarnBlinkTm[4];
			fbBlink.tOffTm	:= tylocalTLBuz.In.tTLWarnBlinkTm[4];
			fbBlink(bEn := TRUE);
			fbWarning(bEn := FALSE);

			tylocalTLBuz.Out.bTLRed		:= tylocalTLBuz.In.bStandby;
			tylocalTLBuz.Out.bTLAmber	:= fbBlink.bOut;
			tylocalTLBuz.Out.bTLGreen	:= tylocalTLBuz.In.bOps;
			tylocalTLBuz.Out.bBuzBeep	:= FALSE;

		ELSIF tylocalTLBuz.In.bWarning[5] = TRUE THEN

			fbBlink.tOnTm	:= tylocalTLBuz.In.tTLWarnBlinkTm[5];
			fbBlink.tOffTm	:= tylocalTLBuz.In.tTLWarnBlinkTm[5];

			fbWarning.tOnTm					:= tylocalTLBuz.In.tBuzWarnOnTm[5]; //Warn T#500ms (from NtParam)
			fbWarning.tOffTm				:= tylocalTLBuz.In.tBuzWarnOnTm[5]; //Warn T#500ms (from NtParam)
			fbWarning.tRstTm				:= tylocalTLBuz.In.tBuzWarnRestTm[5]; //Rest 5 seconds (from NtParam)
			fbWarning.usiOnCnt				:= tylocalTLBuz.In.usiBuzWarnOnCntr[5]; //Count 3 times (from NtParam)
			fbWarning.bStopAftRptSeqEn		:= tylocalTLBuz.In.bBuzWarnStopSeqEn[5]; //Enable Sequence Count (from NtParam)
			fbWarning.usiStopAftRptSeqCntr	:= tylocalTLBuz.In.usiBuzWarnStopSeqCntr[5]; //Sequence Counter  (from NtParam)

			fbBlink(bEn := TRUE);
			fbWarning(bEn := TRUE);

			tylocalTLBuz.Out.bTLRed		:= tylocalTLBuz.In.bStandby;
			tylocalTLBuz.Out.bTLAmber	:= fbBlink.bOut;
			tylocalTLBuz.Out.bTLGreen	:= tylocalTLBuz.In.bOps;
			tylocalTLBuz.Out.bBuzBeep	:= fbWarning.bOut AND (tylocalTLBuz.In.bMuteBuz = FALSE);

		ELSIF tylocalTLBuz.In.bWarningNoBuz[5] = TRUE THEN

			fbBlink.tOnTm	:= tylocalTLBuz.In.tTLWarnBlinkTm[5];
			fbBlink.tOffTm	:= tylocalTLBuz.In.tTLWarnBlinkTm[5];
			fbBlink(bEn := TRUE);
			fbWarning(bEn := FALSE);

			tylocalTLBuz.Out.bTLRed		:= tylocalTLBuz.In.bStandby;
			tylocalTLBuz.Out.bTLAmber	:= fbBlink.bOut;
			tylocalTLBuz.Out.bTLGreen	:= tylocalTLBuz.In.bOps;
			tylocalTLBuz.Out.bBuzBeep	:= FALSE;

		ELSIF tylocalTLBuz.In.bSeqStop = TRUE THEN

			fbBlink.tOnTm	:= tBlinkTm;
			fbBlink.tOffTm	:= tBlinkTm;
			fbBlink(bEn := TRUE);
			fbWarning(bEn := FALSE);

			tylocalTLBuz.Out.bTLRed		:= FALSE;
			tylocalTLBuz.Out.bTLAmber	:= FALSE;
			tylocalTLBuz.Out.bTLGreen	:= fbBlink.bOut;
			tylocalTLBuz.Out.bBuzBeep	:= FALSE;

		ELSIF tylocalTLBuz.In.bChgRcp = TRUE THEN

			fbBlink.tOnTm	:= tylocalTLBuz.In.tTLChgRcpBlinkTm;
			fbBlink.tOffTm	:= tylocalTLBuz.In.tTLChgRcpBlinkTm;
			fbBlink(bEn := TRUE);
			fbWarning(bEn := FALSE);

			IF EDGE(fbBlink.bOut) THEN
				IF tylocalTLBuz.Out.bTLRed = TRUE THEN
					tylocalTLBuz.Out.bTLRed		:= FALSE;
					tylocalTLBuz.Out.bTLAmber	:= FALSE;
					tylocalTLBuz.Out.bTLGreen	:= TRUE;
				ELSIF tylocalTLBuz.Out.bTLAmber = TRUE THEN
					tylocalTLBuz.Out.bTLRed		:= TRUE;
					tylocalTLBuz.Out.bTLAmber	:= FALSE;
					tylocalTLBuz.Out.bTLGreen	:= FALSE;
				ELSE
					tylocalTLBuz.Out.bTLRed		:= FALSE;
					tylocalTLBuz.Out.bTLAmber	:= TRUE;
					tylocalTLBuz.Out.bTLGreen	:= FALSE;
				END_IF
			END_IF

			tylocalTLBuz.Out.bBuzBeep	:= fbBlink.bOut AND (tylocalTLBuz.In.bMuteBuz = FALSE);

		ELSIF tylocalTLBuz.In.bStep = TRUE THEN

			fbBlink.tOnTm	:= tBlinkTm;
			fbBlink.tOffTm	:= tBlinkTm;
			fbBlink(bEn := TRUE);
			fbWarning(bEn := FALSE);

			tylocalTLBuz.Out.bTLRed		:= FALSE;
			tylocalTLBuz.Out.bTLAmber	:= FALSE;
			tylocalTLBuz.Out.bTLGreen	:= fbBlink.bOut;
			tylocalTLBuz.Out.bBuzBeep	:= FALSE;

		ELSIF tylocalTLBuz.In.bOps = TRUE THEN

			fbBlink(bEn := FALSE);
			fbWarning(bEn := FALSE);

			tylocalTLBuz.Out.bTLRed		:= FALSE;
			tylocalTLBuz.Out.bTLAmber	:= FALSE;
			tylocalTLBuz.Out.bTLGreen	:= TRUE;
			tylocalTLBuz.Out.bBuzBeep	:= FALSE;

		ELSIF tylocalTLBuz.In.bSimulation = TRUE THEN

			fbBlink.tOnTm	:= tBlinkTm;
			fbBlink.tOffTm	:= tBlinkTm;
			fbBlink(bEn := TRUE);
			fbWarning(bEn := FALSE);

			tylocalTLBuz.Out.bTLRed		:= fbBlink.bOut;
			tylocalTLBuz.Out.bTLAmber	:= fbBlink.bOut;
			tylocalTLBuz.Out.bTLGreen	:= TRUE;
			tylocalTLBuz.Out.bBuzBeep	:= FALSE;

		ELSIF tylocalTLBuz.In.bStandby = TRUE THEN

			fbBlink(bEn := FALSE);
			fbWarning(bEn := FALSE);

			tylocalTLBuz.Out.bTLRed		:= FALSE;
			tylocalTLBuz.Out.bTLAmber	:= TRUE;
			tylocalTLBuz.Out.bTLGreen	:= FALSE;
			tylocalTLBuz.Out.bBuzBeep	:= FALSE;

		ELSE

			fbBlink(bEn := FALSE);
			fbWarning(bEn := FALSE);

			tylocalTLBuz.Out.bTLRed		:= FALSE;
			tylocalTLBuz.Out.bTLAmber	:= FALSE;
			tylocalTLBuz.Out.bTLGreen	:= FALSE;
			tylocalTLBuz.Out.bBuzBeep	:= FALSE;

		END_IF

	END_IF

	IF tylocalTLBuz.In.bUIManualMod = FALSE AND tylocalTLBuz.In.bErr = FALSE THEN
		IF tylocalTLBuz.In.bTLAmberFlashEn THEN //Amber Flash 1 sec [Put Conditions in Act_Link.st]

			fbBlink1.tOnTm	:= tylocalTLBuz.In.tTLAmberBlinkTm; //T#500ms (from NtParam)
			fbBlink1.tOffTm	:= tylocalTLBuz.In.tTLAmberBlinkTm; //T#500ms (from NtParam)
			fbBlink1(bEn := TRUE);

			tylocalTLBuz.Out.bTLAmber	:= fbBlink1.bOut;

		ELSE
			fbBlink1(bEn := FALSE);
		END_IF

		IF tylocalTLBuz.In.bTLRedFlashEn THEN //Red Flash 1 sec [Put Conditions in Act_Link.st]

			fbBlink2.tOnTm	:= tylocalTLBuz.In.tTLRedBlinkTm; //T#500ms (from NtParam)
			fbBlink2.tOffTm	:= tylocalTLBuz.In.tTLRedBlinkTm; //T#500ms (from NtParam)
			fbBlink2(bEn := TRUE);

			tylocalTLBuz.Out.bTLRed		:= fbBlink2.bOut;
		ELSE
			fbBlink2(bEn := FALSE);
		END_IF

		IF tylocalTLBuz.In.bTLGreenFlashEn THEN //Green Flash 1 sec [Put Conditions in Act_Link.st]

			fbBlink3.tOnTm	:= tylocalTLBuz.In.tTLGreenBlinkTm; //T#500ms (from NtParam)
			fbBlink3.tOffTm	:= tylocalTLBuz.In.tTLGreenBlinkTm; //T#500ms (from NtParam)
			fbBlink3(bEn := TRUE);

			tylocalTLBuz.Out.bTLGreen	:= fbBlink3.bOut;
		ELSE
			fbBlink3(bEn := FALSE);
		END_IF

		IF tylocalTLBuz.In.bBuzAlertEn = TRUE AND fbWarning.bEn=FALSE THEN

			fbWarning1.tOnTm				:= tylocalTLBuz.In.tBuzAlertOnTm;
			fbWarning1.tOffTm				:= tylocalTLBuz.In.tBuzAlertOnTm;
			fbWarning1.tRstTm				:= tylocalTLBuz.In.tBuzAlertRestTm;
			fbWarning1.usiOnCnt				:= tylocalTLBuz.In.usiBuzAlertOnCntr;
			fbWarning1.bStopAftRptSeqEn		:= tylocalTLBuz.In.bBuzAlertStopSeqEn; //Enable Sequence Count (from NtParam)
			fbWarning1.usiStopAftRptSeqCntr	:= tylocalTLBuz.In.usiBuzAlertStopSeqCntr; //Sequence Counter  (from NtParam)

			fbWarning1(bEn := TRUE);

			tylocalTLBuz.Out.bBuzBeep	:= fbWarning1.bOut AND (tylocalTLBuz.In.bMuteBuz = FALSE);

		ELSE
			fbWarning1(bEn := FALSE);
		END_IF
	ELSE
		fbBlink1(bEn := FALSE);
		fbBlink2(bEn := FALSE);
		fbBlink3(bEn := FALSE);
		fbWarning1(bEn := FALSE);
	END_IF

	//Arrange tylocalTLBuz.In.bWarning according to the severity of the warning or info (Err is prioritized)
	IF tylocalTLBuz.In.bErr THEN
		usiWarnInfoStateNew	:= 1;
	ELSIF tylocalTLBuz.In.bWarning[0] THEN
		usiWarnInfoStateNew	:= 2;
	ELSIF tylocalTLBuz.In.bWarning[1] THEN
		usiWarnInfoStateNew	:= 3;
	ELSIF tylocalTLBuz.In.bWarning[2] THEN
		usiWarnInfoStateNew	:= 4;
	ELSIF tylocalTLBuz.In.bWarning[3] THEN
		usiWarnInfoStateNew	:= 5;
	ELSIF tylocalTLBuz.In.bWarning[4] THEN
		usiWarnInfoStateNew	:= 6;
	ELSIF tylocalTLBuz.In.bWarning[5] THEN
		usiWarnInfoStateNew	:= 7;
	ELSIF tylocalTLBuz.In.bBuzAlertEn AND fbWarning.bEn=FALSE THEN
		usiWarnInfoStateNew	:= 8;
	ELSE
		usiWarnInfoStateNew	:= 0;
	END_IF

	IF usiWarnInfoStateOld<>usiWarnInfoStateNew THEN
		usiWarnInfoStateOld:=usiWarnInfoStateNew;
		fbWarning(bEn := FALSE);
		fbWarning1(bEn := FALSE);
	END_IF

END_ACTION
```

#### Act_Background2.st - Do Not Change!!!
```iecst
ACTION Act_Background2: //For MEK machines

	IF EDGEPOS(tylocalTLBuz.In.bUIManualMod) THEN

		fbBlink(bEn := FALSE);
		fbWarning(bEn := FALSE);

		tylocalTLBuz.Out.bTLRed		:= FALSE;
		tylocalTLBuz.Out.bTLAmber	:= TRUE;
		tylocalTLBuz.Out.bTLGreen	:= FALSE;
		tylocalTLBuz.Out.bBuzBeep	:= FALSE;

	ELSIF tylocalTLBuz.In.bUIManualMod THEN

		IF tylocalTLBuz.In.bErr = TRUE THEN

			fbBlink.tOnTm	:= tylocalTLBuz.In.tTLErrBlinkTm; //Error T#500ms (from NtParam)
			fbBlink.tOffTm	:= tylocalTLBuz.In.tTLErrBlinkTm; //Error T#500ms (from NtParam)

			fbWarning.tOnTm					:= tylocalTLBuz.In.tBuzErrOnTm; //Warn T#500ms (from NtParam)
			fbWarning.tOffTm				:= tylocalTLBuz.In.tBuzErrOnTm; //Warn T#500ms (from NtParam)
			fbWarning.tRstTm				:= tylocalTLBuz.In.tBuzErrRestTm; //Rest 5 seconds (from NtParam)
			fbWarning.usiOnCnt				:= tylocalTLBuz.In.usiBuzErrOnCntr; //Count 3 times (from NtParam)
			fbWarning.bStopAftRptSeqEn		:= tylocalTLBuz.In.bBuzErrStopSeqEn; //Enable Sequence Count (from NtParam)
			fbWarning.usiStopAftRptSeqCntr	:= tylocalTLBuz.In.usiBuzErrStopSeqCntr; //Sequence Counter  (from NtParam)

			fbBlink(bEn := TRUE);
			fbWarning(bEn := TRUE);

			tylocalTLBuz.Out.bTLRed		:= fbBlink.bOut;
			tylocalTLBuz.Out.bBuzBeep	:= (fbWarning.bOut) AND (tylocalTLBuz.In.bMuteBuz = FALSE);

			bManualErrOn := TRUE;

		ELSIF bManualErrOn THEN

			fbBlink(bEn := FALSE);
			fbWarning(bEn := FALSE);

			tylocalTLBuz.Out.bTLRed		:= FALSE;
			tylocalTLBuz.Out.bBuzBeep	:= FALSE;

			bManualErrOn := FALSE;

		END_IF

	ELSIF tylocalTLBuz.In.bUIManualMod = FALSE THEN

		bManualErrOn := FALSE;

		IF tylocalTLBuz.In.bStartup = TRUE THEN

			fbBlink(bEn := FALSE);
			fbWarning(bEn := FALSE);

			tylocalTLBuz.Out.bTLRed		:= TRUE;
			tylocalTLBuz.Out.bTLAmber	:= TRUE;
			tylocalTLBuz.Out.bTLGreen	:= TRUE;
			tylocalTLBuz.Out.bBuzBeep	:= FALSE;

		ELSIF tylocalTLBuz.In.bErr = TRUE THEN

			fbBlink.tOnTm	:= tylocalTLBuz.In.tTLErrBlinkTm; //Error T#500ms (from NtParam)
			fbBlink.tOffTm	:= tylocalTLBuz.In.tTLErrBlinkTm; //Error T#500ms (from NtParam)

			fbWarning.tOnTm					:= tylocalTLBuz.In.tBuzErrOnTm; //Warn T#500ms (from NtParam)
			fbWarning.tOffTm				:= tylocalTLBuz.In.tBuzErrOnTm; //Warn T#500ms (from NtParam)
			fbWarning.tRstTm				:= tylocalTLBuz.In.tBuzErrRestTm; //Rest 5 seconds (from NtParam)
			fbWarning.usiOnCnt				:= tylocalTLBuz.In.usiBuzErrOnCntr; //Count 3 times (from NtParam)
			fbWarning.bStopAftRptSeqEn		:= tylocalTLBuz.In.bBuzErrStopSeqEn; //Enable Sequence Count (from NtParam)
			fbWarning.usiStopAftRptSeqCntr	:= tylocalTLBuz.In.usiBuzErrStopSeqCntr; //Sequence Counter  (from NtParam)

			fbBlink(bEn := TRUE);
			fbWarning(bEn := TRUE);

			tylocalTLBuz.Out.bTLRed		:= fbBlink.bOut;
			tylocalTLBuz.Out.bTLAmber	:= FALSE;
			tylocalTLBuz.Out.bTLGreen	:= FALSE;
			tylocalTLBuz.Out.bBuzBeep	:= (fbWarning.bOut) AND (tylocalTLBuz.In.bMuteBuz = FALSE);

		ELSIF tylocalTLBuz.In.bErrNoBuz = TRUE THEN

			fbBlink.tOnTm	:= tylocalTLBuz.In.tTLErrBlinkTm;
			fbBlink.tOffTm	:= tylocalTLBuz.In.tTLErrBlinkTm;
			fbBlink(bEn := TRUE);
			fbWarning(bEn := FALSE);

			tylocalTLBuz.Out.bTLRed		:= fbBlink.bOut;
			tylocalTLBuz.Out.bTLAmber	:= FALSE;
			tylocalTLBuz.Out.bTLGreen	:= FALSE;
			tylocalTLBuz.Out.bBuzBeep	:= FALSE;

		ELSIF tylocalTLBuz.In.bOps = TRUE AND tylocalTLBuz.In.bAOIErrSig = TRUE AND tylocalTLBuz.In.bAOIOriginSig = FALSE THEN

			fbBlink.tOnTm	:= tylocalTLBuz.In.tTLErrBlinkTm;
			fbBlink.tOffTm	:= tylocalTLBuz.In.tTLErrBlinkTm;
			fbBlink(bEn := TRUE);
			fbWarning(bEn := FALSE);

			tylocalTLBuz.Out.bTLRed		:= fbBlink.bOut;
			tylocalTLBuz.Out.bTLAmber	:= FALSE;
			tylocalTLBuz.Out.bTLGreen	:= FALSE;
			tylocalTLBuz.Out.bBuzBeep	:= (fbBlink.bOut) AND (tylocalTLBuz.In.bMuteBuz = FALSE);

		ELSIF tylocalTLBuz.In.bOps = TRUE AND tylocalTLBuz.In.bAOIErrSig = TRUE AND tylocalTLBuz.In.bAOIOriginSig = TRUE THEN

			fbBlink.tOnTm	:= tylocalTLBuz.In.tTLErrBlinkTm;
			fbBlink.tOffTm	:= tylocalTLBuz.In.tTLErrBlinkTm;
			fbBlink(bEn := TRUE);
			fbWarning(bEn := FALSE);

			tylocalTLBuz.Out.bTLRed		:= fbBlink.bOut;
			tylocalTLBuz.Out.bTLAmber	:= FALSE;
			tylocalTLBuz.Out.bTLGreen	:= TRUE;
			tylocalTLBuz.Out.bBuzBeep	:= (fbBlink.bOut) AND (tylocalTLBuz.In.bMuteBuz = FALSE);

		ELSIF tylocalTLBuz.In.bWarning[0] = TRUE THEN

			fbBlink.tOnTm	:= tylocalTLBuz.In.tTLWarnBlinkTm[0]; //Warn T#500ms (from NtParam)
			fbBlink.tOffTm	:= tylocalTLBuz.In.tTLWarnBlinkTm[0]; //Warn T#500ms (from NtParam)

			fbWarning.tOnTm					:= tylocalTLBuz.In.tBuzWarnOnTm[0]; //Warn T#500ms (from NtParam)
			fbWarning.tOffTm				:= tylocalTLBuz.In.tBuzWarnOnTm[0]; //Warn T#500ms (from NtParam)
			fbWarning.tRstTm				:= tylocalTLBuz.In.tBuzWarnRestTm[0]; //Rest 5 seconds (from NtParam)
			fbWarning.usiOnCnt				:= tylocalTLBuz.In.usiBuzWarnOnCntr[0]; //Count 3 times (from NtParam)
			fbWarning.bStopAftRptSeqEn		:= tylocalTLBuz.In.bBuzWarnStopSeqEn[0]; //Enable Sequence Count (from NtParam)
			fbWarning.usiStopAftRptSeqCntr	:= tylocalTLBuz.In.usiBuzWarnStopSeqCntr[0]; //Sequence Counter  (from NtParam)

			fbBlink(bEn := TRUE);
			fbWarning(bEn := TRUE);

			tylocalTLBuz.Out.bTLRed		:= tylocalTLBuz.In.bStandby;
			tylocalTLBuz.Out.bTLAmber	:= fbBlink.bOut;
			tylocalTLBuz.Out.bTLGreen	:= tylocalTLBuz.In.bOps;
			tylocalTLBuz.Out.bBuzBeep	:= fbWarning.bOut AND (tylocalTLBuz.In.bMuteBuz = FALSE);

		ELSIF tylocalTLBuz.In.bWarningNoBuz[0] = TRUE THEN

			fbBlink.tOnTm	:= tylocalTLBuz.In.tTLWarnBlinkTm[0];
			fbBlink.tOffTm	:= tylocalTLBuz.In.tTLWarnBlinkTm[0];
			fbBlink(bEn := TRUE);
			fbWarning(bEn := FALSE);

			tylocalTLBuz.Out.bTLRed		:= tylocalTLBuz.In.bStandby;
			tylocalTLBuz.Out.bTLAmber	:= fbBlink.bOut;
			tylocalTLBuz.Out.bTLGreen	:= tylocalTLBuz.In.bOps;
			tylocalTLBuz.Out.bBuzBeep	:= FALSE;

		ELSIF tylocalTLBuz.In.bWarning[1] = TRUE THEN

			fbBlink.tOnTm	:= tylocalTLBuz.In.tTLWarnBlinkTm[1];
			fbBlink.tOffTm	:= tylocalTLBuz.In.tTLWarnBlinkTm[1];

			fbWarning.tOnTm					:= tylocalTLBuz.In.tBuzWarnOnTm[1]; //Warn T#500ms (from NtParam)
			fbWarning.tOffTm				:= tylocalTLBuz.In.tBuzWarnOnTm[1]; //Warn T#500ms (from NtParam)
			fbWarning.tRstTm				:= tylocalTLBuz.In.tBuzWarnRestTm[1]; //Rest 5 seconds (from NtParam)
			fbWarning.usiOnCnt				:= tylocalTLBuz.In.usiBuzWarnOnCntr[1]; //Count 3 times (from NtParam)
			fbWarning.bStopAftRptSeqEn		:= tylocalTLBuz.In.bBuzWarnStopSeqEn[1]; //Enable Sequence Count (from NtParam)
			fbWarning.usiStopAftRptSeqCntr	:= tylocalTLBuz.In.usiBuzWarnStopSeqCntr[1]; //Sequence Counter  (from NtParam)

			fbBlink(bEn := TRUE);
			fbWarning(bEn := TRUE);

			tylocalTLBuz.Out.bTLRed		:= tylocalTLBuz.In.bStandby;
			tylocalTLBuz.Out.bTLAmber	:= fbBlink.bOut;
			tylocalTLBuz.Out.bTLGreen	:= tylocalTLBuz.In.bOps;
			tylocalTLBuz.Out.bBuzBeep	:= fbWarning.bOut AND (tylocalTLBuz.In.bMuteBuz = FALSE);

		ELSIF tylocalTLBuz.In.bWarningNoBuz[1] = TRUE THEN

			fbBlink.tOnTm	:= tylocalTLBuz.In.tTLWarnBlinkTm[1];
			fbBlink.tOffTm	:= tylocalTLBuz.In.tTLWarnBlinkTm[1];
			fbBlink(bEn := TRUE);
			fbWarning(bEn := FALSE);

			tylocalTLBuz.Out.bTLRed		:= tylocalTLBuz.In.bStandby;
			tylocalTLBuz.Out.bTLAmber	:= fbBlink.bOut;
			tylocalTLBuz.Out.bTLGreen	:= tylocalTLBuz.In.bOps;
			tylocalTLBuz.Out.bBuzBeep	:= FALSE;

		ELSIF tylocalTLBuz.In.bWarning[2] = TRUE THEN

			fbBlink.tOnTm	:= tylocalTLBuz.In.tTLWarnBlinkTm[2];
			fbBlink.tOffTm	:= tylocalTLBuz.In.tTLWarnBlinkTm[2];

			fbWarning.tOnTm					:= tylocalTLBuz.In.tBuzWarnOnTm[2]; //Warn T#500ms (from NtParam)
			fbWarning.tOffTm				:= tylocalTLBuz.In.tBuzWarnOnTm[2]; //Warn T#500ms (from NtParam)
			fbWarning.tRstTm				:= tylocalTLBuz.In.tBuzWarnRestTm[2]; //Rest 5 seconds (from NtParam)
			fbWarning.usiOnCnt				:= tylocalTLBuz.In.usiBuzWarnOnCntr[2]; //Count 3 times (from NtParam)
			fbWarning.bStopAftRptSeqEn		:= tylocalTLBuz.In.bBuzWarnStopSeqEn[2]; //Enable Sequence Count (from NtParam)
			fbWarning.usiStopAftRptSeqCntr	:= tylocalTLBuz.In.usiBuzWarnStopSeqCntr[2]; //Sequence Counter  (from NtParam)

			fbBlink(bEn := TRUE);
			fbWarning(bEn := TRUE);

			tylocalTLBuz.Out.bTLRed		:= tylocalTLBuz.In.bStandby;
			tylocalTLBuz.Out.bTLAmber	:= fbBlink.bOut;
			tylocalTLBuz.Out.bTLGreen	:= tylocalTLBuz.In.bOps;
			tylocalTLBuz.Out.bBuzBeep	:= fbWarning.bOut AND (tylocalTLBuz.In.bMuteBuz = FALSE);

		ELSIF tylocalTLBuz.In.bWarningNoBuz[2] = TRUE THEN

			fbBlink.tOnTm	:= tylocalTLBuz.In.tTLWarnBlinkTm[2];
			fbBlink.tOffTm	:= tylocalTLBuz.In.tTLWarnBlinkTm[2];
			fbBlink(bEn := TRUE);
			fbWarning(bEn := FALSE);

			tylocalTLBuz.Out.bTLRed		:= tylocalTLBuz.In.bStandby;
			tylocalTLBuz.Out.bTLAmber	:= fbBlink.bOut;
			tylocalTLBuz.Out.bTLGreen	:= tylocalTLBuz.In.bOps;
			tylocalTLBuz.Out.bBuzBeep	:= FALSE;

		ELSIF tylocalTLBuz.In.bWarning[3] = TRUE THEN

			fbBlink.tOnTm	:= tylocalTLBuz.In.tTLWarnBlinkTm[3];
			fbBlink.tOffTm	:= tylocalTLBuz.In.tTLWarnBlinkTm[3];

			fbWarning.tOnTm					:= tylocalTLBuz.In.tBuzWarnOnTm[3]; //Warn T#500ms (from NtParam)
			fbWarning.tOffTm				:= tylocalTLBuz.In.tBuzWarnOnTm[3]; //Warn T#500ms (from NtParam)
			fbWarning.tRstTm				:= tylocalTLBuz.In.tBuzWarnRestTm[3]; //Rest 5 seconds (from NtParam)
			fbWarning.usiOnCnt				:= tylocalTLBuz.In.usiBuzWarnOnCntr[3]; //Count 3 times (from NtParam)
			fbWarning.bStopAftRptSeqEn		:= tylocalTLBuz.In.bBuzWarnStopSeqEn[3]; //Enable Sequence Count (from NtParam)
			fbWarning.usiStopAftRptSeqCntr	:= tylocalTLBuz.In.usiBuzWarnStopSeqCntr[3]; //Sequence Counter  (from NtParam)

			fbBlink(bEn := TRUE);
			fbWarning(bEn := TRUE);

			tylocalTLBuz.Out.bTLRed		:= tylocalTLBuz.In.bStandby;
			tylocalTLBuz.Out.bTLAmber	:= fbBlink.bOut;
			tylocalTLBuz.Out.bTLGreen	:= tylocalTLBuz.In.bOps;
			tylocalTLBuz.Out.bBuzBeep	:= fbWarning.bOut AND (tylocalTLBuz.In.bMuteBuz = FALSE);

		ELSIF tylocalTLBuz.In.bWarningNoBuz[3] = TRUE THEN

			fbBlink.tOnTm	:= tylocalTLBuz.In.tTLWarnBlinkTm[3];
			fbBlink.tOffTm	:= tylocalTLBuz.In.tTLWarnBlinkTm[3];
			fbBlink(bEn := TRUE);
			fbWarning(bEn := FALSE);

			tylocalTLBuz.Out.bTLRed		:= tylocalTLBuz.In.bStandby;
			tylocalTLBuz.Out.bTLAmber	:= fbBlink.bOut;
			tylocalTLBuz.Out.bTLGreen	:= tylocalTLBuz.In.bOps;
			tylocalTLBuz.Out.bBuzBeep	:= FALSE;

		ELSIF tylocalTLBuz.In.bWarning[4] = TRUE THEN

			fbBlink.tOnTm	:= tylocalTLBuz.In.tTLWarnBlinkTm[4];
			fbBlink.tOffTm	:= tylocalTLBuz.In.tTLWarnBlinkTm[4];

			fbWarning.tOnTm					:= tylocalTLBuz.In.tBuzWarnOnTm[4]; //Warn T#500ms (from NtParam)
			fbWarning.tOffTm				:= tylocalTLBuz.In.tBuzWarnOnTm[4]; //Warn T#500ms (from NtParam)
			fbWarning.tRstTm				:= tylocalTLBuz.In.tBuzWarnRestTm[4]; //Rest 5 seconds (from NtParam)
			fbWarning.usiOnCnt				:= tylocalTLBuz.In.usiBuzWarnOnCntr[4]; //Count 3 times (from NtParam)
			fbWarning.bStopAftRptSeqEn		:= tylocalTLBuz.In.bBuzWarnStopSeqEn[4]; //Enable Sequence Count (from NtParam)
			fbWarning.usiStopAftRptSeqCntr	:= tylocalTLBuz.In.usiBuzWarnStopSeqCntr[4]; //Sequence Counter  (from NtParam)

			fbBlink(bEn := TRUE);
			fbWarning(bEn := TRUE);

			tylocalTLBuz.Out.bTLRed		:= tylocalTLBuz.In.bStandby;
			tylocalTLBuz.Out.bTLAmber	:= fbBlink.bOut;
			tylocalTLBuz.Out.bTLGreen	:= tylocalTLBuz.In.bOps;
			tylocalTLBuz.Out.bBuzBeep	:= fbWarning.bOut AND (tylocalTLBuz.In.bMuteBuz = FALSE);

		ELSIF tylocalTLBuz.In.bWarningNoBuz[4] = TRUE THEN

			fbBlink.tOnTm	:= tylocalTLBuz.In.tTLWarnBlinkTm[4];
			fbBlink.tOffTm	:= tylocalTLBuz.In.tTLWarnBlinkTm[4];
			fbBlink(bEn := TRUE);
			fbWarning(bEn := FALSE);

			tylocalTLBuz.Out.bTLRed		:= tylocalTLBuz.In.bStandby;
			tylocalTLBuz.Out.bTLAmber	:= fbBlink.bOut;
			tylocalTLBuz.Out.bTLGreen	:= tylocalTLBuz.In.bOps;
			tylocalTLBuz.Out.bBuzBeep	:= FALSE;

		ELSIF tylocalTLBuz.In.bWarning[5] = TRUE THEN

			fbBlink.tOnTm	:= tylocalTLBuz.In.tTLWarnBlinkTm[5];
			fbBlink.tOffTm	:= tylocalTLBuz.In.tTLWarnBlinkTm[5];

			fbWarning.tOnTm					:= tylocalTLBuz.In.tBuzWarnOnTm[5]; //Warn T#500ms (from NtParam)
			fbWarning.tOffTm				:= tylocalTLBuz.In.tBuzWarnOnTm[5]; //Warn T#500ms (from NtParam)
			fbWarning.tRstTm				:= tylocalTLBuz.In.tBuzWarnRestTm[5]; //Rest 5 seconds (from NtParam)
			fbWarning.usiOnCnt				:= tylocalTLBuz.In.usiBuzWarnOnCntr[5]; //Count 3 times (from NtParam)
			fbWarning.bStopAftRptSeqEn		:= tylocalTLBuz.In.bBuzWarnStopSeqEn[5]; //Enable Sequence Count (from NtParam)
			fbWarning.usiStopAftRptSeqCntr	:= tylocalTLBuz.In.usiBuzWarnStopSeqCntr[5]; //Sequence Counter  (from NtParam)

			fbBlink(bEn := TRUE);
			fbWarning(bEn := TRUE);

			tylocalTLBuz.Out.bTLRed		:= tylocalTLBuz.In.bStandby;
			tylocalTLBuz.Out.bTLAmber	:= fbBlink.bOut;
			tylocalTLBuz.Out.bTLGreen	:= tylocalTLBuz.In.bOps;
			tylocalTLBuz.Out.bBuzBeep	:= fbWarning.bOut AND (tylocalTLBuz.In.bMuteBuz = FALSE);

		ELSIF tylocalTLBuz.In.bWarningNoBuz[5] = TRUE THEN

			fbBlink.tOnTm	:= tylocalTLBuz.In.tTLWarnBlinkTm[5];
			fbBlink.tOffTm	:= tylocalTLBuz.In.tTLWarnBlinkTm[5];
			fbBlink(bEn := TRUE);
			fbWarning(bEn := FALSE);

			tylocalTLBuz.Out.bTLRed		:= tylocalTLBuz.In.bStandby;
			tylocalTLBuz.Out.bTLAmber	:= fbBlink.bOut;
			tylocalTLBuz.Out.bTLGreen	:= tylocalTLBuz.In.bOps;
			tylocalTLBuz.Out.bBuzBeep	:= FALSE;

		ELSIF tylocalTLBuz.In.bSeqStop = TRUE THEN

			fbBlink.tOnTm	:= tBlinkTm;
			fbBlink.tOffTm	:= tBlinkTm;
			fbBlink(bEn := TRUE);
			fbWarning(bEn := FALSE);

			tylocalTLBuz.Out.bTLRed		:= fbBlink.bOut;
			tylocalTLBuz.Out.bTLAmber	:= FALSE;
			tylocalTLBuz.Out.bTLGreen	:= TRUE;
			tylocalTLBuz.Out.bBuzBeep	:= FALSE;

		ELSIF tylocalTLBuz.In.bChgRcp = TRUE THEN

			fbBlink.tOnTm	:= tylocalTLBuz.In.tTLChgRcpBlinkTm;
			fbBlink.tOffTm	:= tylocalTLBuz.In.tTLChgRcpBlinkTm;
			fbBlink(bEn := TRUE);
			fbWarning(bEn := FALSE);

			IF EDGE(fbBlink.bOut) THEN
				IF tylocalTLBuz.Out.bTLRed = TRUE THEN
					tylocalTLBuz.Out.bTLRed		:= FALSE;
					tylocalTLBuz.Out.bTLAmber	:= FALSE;
					tylocalTLBuz.Out.bTLGreen	:= TRUE;
				ELSIF tylocalTLBuz.Out.bTLAmber = TRUE THEN
					tylocalTLBuz.Out.bTLRed		:= TRUE;
					tylocalTLBuz.Out.bTLAmber	:= FALSE;
					tylocalTLBuz.Out.bTLGreen	:= FALSE;
				ELSE
					tylocalTLBuz.Out.bTLRed		:= FALSE;
					tylocalTLBuz.Out.bTLAmber	:= TRUE;
					tylocalTLBuz.Out.bTLGreen	:= FALSE;
				END_IF
			END_IF

			tylocalTLBuz.Out.bBuzBeep	:= fbBlink.bOut AND (tylocalTLBuz.In.bMuteBuz = FALSE);

		ELSIF tylocalTLBuz.In.bStep = TRUE THEN

			fbBlink.tOnTm	:= tBlinkTm;
			fbBlink.tOffTm	:= tBlinkTm;
			fbBlink(bEn := TRUE);
			fbWarning(bEn := FALSE);

			tylocalTLBuz.Out.bTLRed		:= FALSE;
			tylocalTLBuz.Out.bTLAmber	:= FALSE;
			tylocalTLBuz.Out.bTLGreen	:= fbBlink.bOut;
			tylocalTLBuz.Out.bBuzBeep	:= FALSE;

		ELSIF tylocalTLBuz.In.bOps = TRUE THEN

			fbBlink(bEn := FALSE);
			fbWarning(bEn := FALSE);

			tylocalTLBuz.Out.bTLRed		:= FALSE;
			tylocalTLBuz.Out.bTLAmber	:= FALSE;
			tylocalTLBuz.Out.bTLGreen	:= TRUE;
			tylocalTLBuz.Out.bBuzBeep	:= FALSE;

		ELSIF tylocalTLBuz.In.bSimulation = TRUE THEN

			fbBlink.tOnTm	:= tBlinkTm;
			fbBlink.tOffTm	:= tBlinkTm;
			fbBlink(bEn := TRUE);
			fbWarning(bEn := FALSE);

			tylocalTLBuz.Out.bTLRed		:= fbBlink.bOut;
			tylocalTLBuz.Out.bTLAmber	:= fbBlink.bOut;
			tylocalTLBuz.Out.bTLGreen	:= TRUE;
			tylocalTLBuz.Out.bBuzBeep	:= FALSE;

		ELSIF tylocalTLBuz.In.bStandby = TRUE THEN

			fbBlink(bEn := FALSE);
			fbWarning(bEn := FALSE);

			tylocalTLBuz.Out.bTLRed		:= TRUE;
			tylocalTLBuz.Out.bTLAmber	:= FALSE;
			tylocalTLBuz.Out.bTLGreen	:= FALSE;
			tylocalTLBuz.Out.bBuzBeep	:= FALSE;

		ELSE

			fbBlink(bEn := FALSE);
			fbWarning(bEn := FALSE);

			tylocalTLBuz.Out.bTLRed		:= FALSE;
			tylocalTLBuz.Out.bTLAmber	:= FALSE;
			tylocalTLBuz.Out.bTLGreen	:= FALSE;
			tylocalTLBuz.Out.bBuzBeep	:= FALSE;

		END_IF

	END_IF

	IF tylocalTLBuz.In.bUIManualMod = FALSE AND tylocalTLBuz.In.bErr = FALSE THEN
		IF tylocalTLBuz.In.bTLAmberFlashEn THEN //Amber Flash 1 sec [Put Conditions in Act_Link.st]

			fbBlink1.tOnTm	:= tylocalTLBuz.In.tTLAmberBlinkTm; //T#500ms (from NtParam)
			fbBlink1.tOffTm	:= tylocalTLBuz.In.tTLAmberBlinkTm; //T#500ms (from NtParam)
			fbBlink1(bEn := TRUE);

			tylocalTLBuz.Out.bTLAmber	:= fbBlink1.bOut;

		ELSE
			fbBlink1(bEn := FALSE);
		END_IF

		IF tylocalTLBuz.In.bTLRedFlashEn THEN //Red Flash 1 sec [Put Conditions in Act_Link.st]

			fbBlink2.tOnTm	:= tylocalTLBuz.In.tTLRedBlinkTm; //T#500ms (from NtParam)
			fbBlink2.tOffTm	:= tylocalTLBuz.In.tTLRedBlinkTm; //T#500ms (from NtParam)
			fbBlink2(bEn := TRUE);

			tylocalTLBuz.Out.bTLRed		:= fbBlink2.bOut;
		ELSE
			fbBlink2(bEn := FALSE);
		END_IF

		IF tylocalTLBuz.In.bTLGreenFlashEn THEN //Green Flash 1 sec [Put Conditions in Act_Link.st]

			fbBlink3.tOnTm	:= tylocalTLBuz.In.tTLGreenBlinkTm; //T#500ms (from NtParam)
			fbBlink3.tOffTm	:= tylocalTLBuz.In.tTLGreenBlinkTm; //T#500ms (from NtParam)
			fbBlink3(bEn := TRUE);

			tylocalTLBuz.Out.bTLGreen	:= fbBlink3.bOut;
		ELSE
			fbBlink3(bEn := FALSE);
		END_IF

		IF tylocalTLBuz.In.bBuzAlertEn = TRUE AND fbWarning.bEn=FALSE THEN

			fbWarning1.tOnTm				:= tylocalTLBuz.In.tBuzAlertOnTm;
			fbWarning1.tOffTm				:= tylocalTLBuz.In.tBuzAlertOnTm;
			fbWarning1.tRstTm				:= tylocalTLBuz.In.tBuzAlertRestTm;
			fbWarning1.usiOnCnt				:= tylocalTLBuz.In.usiBuzAlertOnCntr;
			fbWarning1.bStopAftRptSeqEn		:= tylocalTLBuz.In.bBuzAlertStopSeqEn; //Enable Sequence Count (from NtParam)
			fbWarning1.usiStopAftRptSeqCntr	:= tylocalTLBuz.In.usiBuzAlertStopSeqCntr; //Sequence Counter  (from NtParam)

			fbWarning1(bEn := TRUE);

			tylocalTLBuz.Out.bBuzBeep	:= fbWarning1.bOut AND (tylocalTLBuz.In.bMuteBuz = FALSE);

		ELSE
			fbWarning1(bEn := FALSE);
		END_IF
	ELSE
		fbBlink1(bEn := FALSE);
		fbBlink2(bEn := FALSE);
		fbBlink3(bEn := FALSE);
		fbWarning1(bEn := FALSE);
	END_IF

	//Arrange tylocalTLBuz.In.bWarning according to the severity of the warning or info (Err is prioritized)
	IF tylocalTLBuz.In.bErr THEN
		usiWarnInfoStateNew	:= 1;
	ELSIF tylocalTLBuz.In.bWarning[0] THEN
		usiWarnInfoStateNew	:= 2;
	ELSIF tylocalTLBuz.In.bWarning[1] THEN
		usiWarnInfoStateNew	:= 3;
	ELSIF tylocalTLBuz.In.bWarning[2] THEN
		usiWarnInfoStateNew	:= 4;
	ELSIF tylocalTLBuz.In.bWarning[3] THEN
		usiWarnInfoStateNew	:= 5;
	ELSIF tylocalTLBuz.In.bWarning[4] THEN
		usiWarnInfoStateNew	:= 6;
	ELSIF tylocalTLBuz.In.bWarning[5] THEN
		usiWarnInfoStateNew	:= 7;
	ELSIF tylocalTLBuz.In.bBuzAlertEn AND fbWarning.bEn=FALSE THEN
		usiWarnInfoStateNew	:= 8;
	ELSE
		usiWarnInfoStateNew	:= 0;
	END_IF

	IF usiWarnInfoStateOld<>usiWarnInfoStateNew THEN
		usiWarnInfoStateOld:=usiWarnInfoStateNew;
		fbWarning(bEn := FALSE);
		fbWarning1(bEn := FALSE);
	END_IF

END_ACTION
```
